//电流超限监测
FOR i:=1 TO g_maxCartJoint BY 1 DO
	m_checkDelay[i_armId].T_cartJntCurrentErr[i](IN:= ABS(i_cartJointData.m_curJntTrq[i])>g_cartMaxJntCurrent[i] AND m_checkPermit[i_ArmId].m_cartJntCurrentErr[i], PT:=m_checkDelayTime.Ti_CarJntCurrent , Q=> , ET=> );
	IF m_checkDelay[i_armId].T_cartJntCurrentErr[i].Q THEN
		errCodeAssign(i_armId, i_ArmId,  0, i, 16#2005 ,m_rcvLevel );
	END_IF
END_FOR


//Ethercat通讯检测
FOR i:=1 TO g_maxCartJoint BY 1 DO
	IF NOT i_safetyCheckVar.m_cartEtherCATState[i].EtherCATState THEN
		errCodeAssign(i_armId, i_ArmId,  0, i, 16#2006 ,m_rcvLevel );
	END_IF
END_FOR
END_METHOD

PROPERTY checkPermit : REFERENCE TO ARRAY[1..g_maxNum] OF  checkPermit
GET
checkPermit ref= m_checkPermit;
END_GET
SET
END_SET
END_PROPERTY

METHOD electriAngleDev : DINT
VAR_INPUT
	i_motorElectriAngleDev : DINT;
END_VAR

IF i_motorElectriAngleDev > 50000 THEN
	electriAngleDev := i_motorElectriAngleDev - 65535;
ELSIF i_motorElectriAngleDev < -50000 THEN
	electriAngleDev := i_motorElectriAngleDev + 65535;
ELSE
	electriAngleDev := i_motorElectriAngleDev;
END_IF
END_METHOD

METHOD errCodeAssign : BOOL
VAR_INPUT
	i_armId:UDINT;
	i_errLocation:UDINT;
	i_errCodeMode:UDINT;
	i_errJoint:UDINT;
	i_errID:UDINT;
	i_errFlagID :UINT;
END_VAR
IF m_jntErrFlag[i_armId,i_errJoint,i_errFlagID]=FALSE THEN
	m_jntErrFlag[i_armId,i_errJoint,i_errFlagID]:=TRUE;
	m_errCode:=SHL(i_errLocation,24)+SHL(i_errCodeMode,20)+SHL(i_errJoint,16)+i_errID;
	
	
	IF i_errID>=16#3000 THEN
		m_errNumType[m_unrcvLevel]:=LIMIT(0,m_errNumType[m_unrcvLevel]+1,100);
		m_arrayErrCodeType[m_unrcvLevel][m_errNumType[m_unrcvLevel]]:=m_errCode;
		g_arrayErrCodeArm[i_armId]:=arrayFILO(i_Array:= g_arrayErrCodeArm[i_ArmId], i_NewData:=m_errCode );
		m_armErrFlag[i_armId,m_unrcvLevel]:=TRUE;
		
	ELSIF i_errID>=16#2000 THEN
		m_errNumType[m_rcvLevel]:=LIMIT(0,m_errNumType[m_rcvLevel]+1,100);
		m_arrayErrCodeType[m_rcvLevel][m_errNumType[m_rcvLevel]]:=m_errCode;
		g_arrayErrCodeArm[i_armId]:=arrayFILO(i_Array:= g_arrayErrCodeArm[i_ArmId], i_NewData:=m_errCode );
		m_armErrFlag[i_armId,m_rcvLevel]:=TRUE;
		
	END_IF
END_IF
END_METHOD

METHOD errCodeUpdating :ARRAY [1..3] OF UDINT;
VAR_INPUT
END_VAR

m_errCodeUpdateTon[m_unrcvLevel](IN:= NOT m_errCodeUpdateFlag[3], PT:=m_codeUpdateDelay , Q=> m_errCodeUpdateFlag[3], ET=> );
IF m_errCodeUpdateFlag[m_unrcvLevel] THEN
	IF m_errNumType[m_unrcvLevel]>=1 THEN
		m_ArrayErrCodeType[m_unrcvLevel]:=ArrayDeleteFrist(i_Array:=m_ArrayErrCodeType[3]) ;
		o_ErrCode[m_unrcvLevel]:=m_ArrayErrCodeType[m_unrcvLevel][0] ;
		m_errNumType[m_unrcvLevel]:=m_errNumType[m_unrcvLevel]-1;
	END_IF
END_IF


m_errCodeUpdateTon[m_rcvLevel](IN:= NOT m_errCodeUpdateFlag[2], PT:=m_codeUpdateDelay , Q=> m_errCodeUpdateFlag[2], ET=> );
IF m_errCodeUpdateFlag[m_rcvLevel] THEN
	IF m_errNumType[m_rcvLevel]>=1 THEN
		m_ArrayErrCodeType[m_rcvLevel]:=ArrayDeleteFrist(i_Array:=m_ArrayErrCodeType[m_rcvLevel]) ;
		o_ErrCode[m_rcvLevel]:=m_ArrayErrCodeType[m_rcvLevel][0] ;
		m_errNumType[m_rcvLevel]:=m_errNumType[m_rcvLevel]-1;
	END_IF
END_IF
END_METHOD

METHOD errFlagReset : BOOL
VAR_INPUT
END_VAR

FOR i := 1 TO g_maxNum DO
	FOR j :=0 TO g_maxArmJoint DO
		m_jntErrFlag[i, j, 2]:=FALSE;
	END_FOR
	m_armErrFlag[i, 2]:=FALSE;
END_FOR

o_ErrCode[2]:=0;
END_METHOD

METHOD poseErrCheck : vec6d
VAR_INPUT
	i_cmdPose : ST_Frame;
	i_curPose :ST_Frame;
END_VAR

VAR
	posErr,oriErr:Vec3d;
	matT,rotErr:Mat3d;
	errAngle :LREAL;
	errAxis :Vec3d;
	i : INT;
END_VAR
vecSub(i_cmdPose.m_pos, i_curPose.m_pos,posErr);

matTranspose(i_cmdPose.m_rot, matT);
matMultiply(matT,i_curPose.m_rot, rotErr);
rot2AngAxis(rotErr, angle=>errAngle, axis=>errAxis);
vecMultiNum(errAxis, errAngle,oriErr);

FOR i := 1 TO 6 DO
	IF i <= 3 THEN
		poseErrCheck[i] := posErr[i];
	ELSE
		poseErrCheck[i] := oriErr[i];
	END_IF
END_FOR
END_METHOD

METHOD promptMassCode : BOOL
VAR_INPUT
	i_PromptStatus:BOOL;
	i_ArmId:UDINT;
	i_ErrID:UDINT;
	i_ErrLocation:UDINT;
END_VAR

m_PromptMassBusy:=TRUE;

//提示置位
IF i_PromptStatus=TRUE AND m_PromptFlag[i_ArmId,i_ErrID]=0 THEN
	m_PromptFlag[i_ArmId,i_ErrID]:=1;
END_IF

//输出提示故障码
IF m_PromptFlag[i_ArmId,i_ErrID]=1 THEN
	m_ErrCode:=SHL(i_ErrLocation,24)+i_ErrID+16#1010;
	m_ArrayErrCodeType[1]:=ArrayFIFO(i_Array:= m_ArrayErrCodeType[1], i_NewData:=m_ErrCode );//m_ErrCode;
	m_PromptFlag[i_ArmId,i_ErrID]:=2;
END_IF

//清除提示故障码
IF m_PromptFlag[i_ArmId,i_ErrID]=2 AND i_PromptStatus=FALSE THEN
	m_deleteCode:=SHL(i_ErrLocation,24)+i_ErrID+16#1010;
	ArrayDeleteInput(i_Array:= m_ArrayErrCodeType[1], i_DeleteCode:=m_deleteCode , o_Array=> m_ArrayErrCodeType[1]);
	m_PromptFlag[i_ArmId,i_ErrID]:=0;
END_IF
o_ErrCode[1]:=m_ArrayErrCodeType[1][0];
m_PromptMassBusy:=FALSE;
END_METHOD

METHOD systemSafetyCheck : BOOL
VAR_INPUT
	i_armId:UDINT;
	i_safetyCheckVar :ARRAY[1..g_maxNum] OF checkInputVariable;
	i_masterStatus :ST_MasterStatus;
	i_cartJointData : ST_CartJointData;
	i_masterJointData : ST_MasterJointData;
END_VAR

VAR
	k:INT;
END_VAR
IF i_armId =g_cartNum THEN 
	//cart safrty check
	cartSafetyCheck(i_armId,i_safetyCheckVar[i_armId],i_cartJointData);
ELSE
	//master arms safety check
	armSafetyCheck(i_armId,i_safetyCheckVar,i_masterStatus,i_masterJointData);
END_IF

//StopButton
IF  i_safetyCheckVar[i_ArmId].PCStopButton=0 OR NOT i_safetyCheckVar[i_ArmId].MasterStopButton OR i_safetyCheckVar[i_ArmId].SlaveStopButton THEN
	errCodeAssign(i_ArmId, 16#0B, 0, 0, 16#2001, m_rcvLevel );
END_IF

//prompt message
FOR i:=1 TO 10 DO
	PromptMassCode( i_safetyCheckVar[i_ArmId].m_promptStatus[i], i_ArmId,  i,  i_safetyCheckVar[i_ArmId].m_promptLocation[i]);
END_FOR
END_METHOD

END_FUNCTION_BLOCK

// ---- SafetyCheck/Fb_dataRecord.TcPOU
FUNCTION_BLOCK Fb_dataRecord 
VAR_INPUT
	
END_VAR
VAR_OUTPUT
END_VAR
VAR
	i,j,k,z,c:UDINT;
	Index:ARRAY[1..g_maxNum] OF INT:=[3(2)];
	m_Index:ARRAY[1..g_maxNum] OF UDINT;
	Err,Arm,Joint,ErrID:UDINT;
	ErrWritingFalg:ARRAY [1..g_maxNum] OF BOOL:=[3(FALSE)];
	ArrayErrCodeTypeLast:ARRAY [1..g_maxNum] OF UDINT;
	sPath: STRING(255);
	mErr:ARRAY [0..MAX_CSV_COLUMNS] OF STRING(255);
	StartRecord:ARRAY[1..g_maxNum] OF R_TRIG;
	RecordCompletion:ARRAY[1..g_maxNum] OF F_TRIG;
	errFlagDelay1s : ARRAY [1..3] OF TON;
	errWritingAllowed : ARRAY [1..3] OF BOOL:=[3(FALSE)];
	
	fbSysTime	: 	GETSYSTEMTIME;
	tFileTime	:	T_FILETIME;  
	
	_tNow,	_tNowBoLin	:	TIMESTRUCT; 
	fbFormat 	: 	FB_FormatString;
	_sPathFormat	: T_MaxString := '%s%d-%d-%d-%d-%d-%d-%s-%s-%s.csv'; 
	
	_iBuffer: UDINT := 1;
		
	StartTime:LREAL;
	
	iZeroRowsData:ARRAY[0..MAX_CSV_ROWS] OF  ARRAY [0..MAX_CSV_COLUMNS] OF STRING(MAX_CSV_FIELD_LENGTH);
	iZeroErrCode:ARRAY [1..g_maxNum] OF ARRAY[0..100] OF UDINT;
	gCSV_Buffer: ARRAY[1..MAX_CSV_RING_BUFFER] OF ST_Buffer;
	mErrNameLocation: ARRAY [1..MAX_CSV_RING_BUFFER,0..MAX_CSV_COLUMNS] OF STRING(MAX_CSV_FIELD_LENGTH);
END_VAR

METHOD armDataCast : BOOL
VAR_IN_OUT CONSTANT
	i_safetyCheckVar :ARRAY[1..g_maxNum] OF checkInputVariable;
	i_masterStatus : ST_masterStatus;
	i_masterJointData : ST_MasterJointData;
END_VAR

FOR i:= 1 TO 2 BY 1 DO
	IF ErrWritingFalg[i] = FALSE THEN
	j:=1;
	//状态机
	gCSV_Buffer[i].aBuffer[Index[i]][j:=j+1]:=LREAL_TO_FMTSTR(i_masterStatus.m_armState[i],0, TRUE);  gCSV_Buffer[i].aBuffer[1][j]:='armMachine';
	
	//link pos
	gCSV_Buffer[i].aBuffer[Index[i]][j:=j+1]:=LREAL_TO_STRING(i_masterJointData.m_curLinkPos[i][1]);   gCSV_Buffer[i].aBuffer[1][j]:='curLinkPosJ1';
	gCSV_Buffer[i].aBuffer[Index[i]][j:=j+1]:=LREAL_TO_STRING(i_masterJointData.m_curLinkPos[i][2]);   gCSV_Buffer[i].aBuffer[1][j]:='curLinkPosJ2';
	gCSV_Buffer[i].aBuffer[Index[i]][j:=j+1]:=LREAL_TO_STRING(i_masterJointData.m_curLinkPos[i][3]);   gCSV_Buffer[i].aBuffer[1][j]:='curLinkPosJ3';
	gCSV_Buffer[i].aBuffer[Index[i]][j:=j+1]:=LREAL_TO_STRING(i_masterJointData.m_curLinkPos[i][4]);   gCSV_Buffer[i].aBuffer[1][j]:='curLinkPosJ4';
	gCSV_Buffer[i].aBuffer[Index[i]][j:=j+1]:=LREAL_TO_STRING(i_masterJointData.m_curLinkPos[i][5]);   gCSV_Buffer[i].aBuffer[1][j]:='curLinkPosJ5';
	gCSV_Buffer[i].aBuffer[Index[i]][j:=j+1]:=LREAL_TO_STRING(i_masterJointData.m_curLinkPos[i][6]);   gCSV_Buffer[i].aBuffer[1][j]:='curLinkPosJ6';
	gCSV_Buffer[i].aBuffer[Index[i]][j:=j+1]:=LREAL_TO_STRING(i_masterJointData.m_curLinkPos[i][7]);   gCSV_Buffer[i].aBuffer[1][j]:='curLinkPosJ7';
	
	//motor pos / curJntPos
	gCSV_Buffer[i].aBuffer[Index[i]][j:=j+1]:=LREAL_TO_STRING(i_masterJointData.m_curJntPos[i][1]);  gCSV_Buffer[i].aBuffer[1][j]:='curJntPosJ1';
	gCSV_Buffer[i].aBuffer[Index[i]][j:=j+1]:=LREAL_TO_STRING(i_masterJointData.m_curJntPos[i][2]);  gCSV_Buffer[i].aBuffer[1][j]:='curJntPosJ2';
	gCSV_Buffer[i].aBuffer[Index[i]][j:=j+1]:=LREAL_TO_STRING(i_masterJointData.m_curJntPos[i][3]);  gCSV_Buffer[i].aBuffer[1][j]:='curJntPosJ3';
	gCSV_Buffer[i].aBuffer[Index[i]][j:=j+1]:=LREAL_TO_STRING(i_masterJointData.m_curJntPos[i][4]);  gCSV_Buffer[i].aBuffer[1][j]:='curJntPosJ4';
	gCSV_Buffer[i].aBuffer[Index[i]][j:=j+1]:=LREAL_TO_STRING(i_masterJointData.m_curJntPos[i][5]); 	gCSV_Buffer[i].aBuffer[1][j]:='curJntPosJ5';
	gCSV_Buffer[i].aBuffer[Index[i]][j:=j+1]:=LREAL_TO_STRING(i_masterJointData.m_curJntPos[i][6]); 	gCSV_Buffer[i].aBuffer[1][j]:='curJntPosJ6';
	gCSV_Buffer[i].aBuffer[Index[i]][j:=j+1]:=LREAL_TO_STRING(i_masterJointData.m_curJntPos[i][7]); 	gCSV_Buffer[i].aBuffer[1][j]:='curJntPosJ7';
	
	
	//target joint position 
	gCSV_Buffer[i].aBuffer[Index[i]][j:=j+1]:=LREAL_TO_STRING(i_masterJointData.m_cmdJntPos[i][1]);  gCSV_Buffer[i].aBuffer[1][j]:='cmdJntPosJ1';
	gCSV_Buffer[i].aBuffer[Index[i]][j:=j+1]:=LREAL_TO_STRING(i_masterJointData.m_cmdJntPos[i][2]);  gCSV_Buffer[i].aBuffer[1][j]:='cmdJntPosJ2';
	gCSV_Buffer[i].aBuffer[Index[i]][j:=j+1]:=LREAL_TO_STRING(i_masterJointData.m_cmdJntPos[i][3]);  gCSV_Buffer[i].aBuffer[1][j]:='cmdJntPosJ3';
	gCSV_Buffer[i].aBuffer[Index[i]][j:=j+1]:=LREAL_TO_STRING(i_masterJointData.m_cmdJntPos[i][4]);  gCSV_Buffer[i].aBuffer[1][j]:='cmdJntPosJ4';
	gCSV_Buffer[i].aBuffer[Index[i]][j:=j+1]:=LREAL_TO_STRING(i_masterJointData.m_cmdJntPos[i][5]);  gCSV_Buffer[i].aBuffer[1][j]:='cmdJntPosJ5';
	gCSV_Buffer[i].aBuffer[Index[i]][j:=j+1]:=LREAL_TO_STRING(i_masterJointData.m_cmdJntPos[i][6]);  gCSV_Buffer[i].aBuffer[1][j]:='cmdJntPosJ6';
	gCSV_Buffer[i].aBuffer[Index[i]][j:=j+1]:=LREAL_TO_STRING(i_masterJointData.m_cmdJntPos[i][7]);  gCSV_Buffer[i].aBuffer[1][j]:='cmdJntPosJ7';
	
	
	//current joint velocity
	gCSV_Buffer[i].aBuffer[Index[i]][j:=j+1]:=LREAL_TO_STRING(i_masterJointData.m_curJntVel[i][1]);  gCSV_Buffer[i].aBuffer[1][j]:='curJntVelJ1';
	gCSV_Buffer[i].aBuffer[Index[i]][j:=j+1]:=LREAL_TO_STRING(i_masterJointData.m_curJntVel[i][2]);  gCSV_Buffer[i].aBuffer[1][j]:='curJntVelJ2';
	gCSV_Buffer[i].aBuffer[Index[i]][j:=j+1]:=LREAL_TO_STRING(i_masterJointData.m_curJntVel[i][3]);  gCSV_Buffer[i].aBuffer[1][j]:='curJntVelJ3';
	gCSV_Buffer[i].aBuffer[Index[i]][j:=j+1]:=LREAL_TO_STRING(i_masterJointData.m_curJntVel[i][4]);  gCSV_Buffer[i].aBuffer[1][j]:='curJntVelJ4';
	gCSV_Buffer[i].aBuffer[Index[i]][j:=j+1]:=LREAL_TO_STRING(i_masterJointData.m_curJntVel[i][5]);  gCSV_Buffer[i].aBuffer[1][j]:='curJntVelJ5';
	gCSV_Buffer[i].aBuffer[Index[i]][j:=j+1]:=LREAL_TO_STRING(i_masterJointData.m_curJntVel[i][6]);  gCSV_Buffer[i].aBuffer[1][j]:='curJntVelJ6';
	gCSV_Buffer[i].aBuffer[Index[i]][j:=j+1]:=LREAL_TO_STRING(i_masterJointData.m_curJntVel[i][7]);  gCSV_Buffer[i].aBuffer[1][j]:='curJntVelJ7';
	
	//command arm pose
	gCSV_Buffer[i].aBuffer[Index[i]][j:=j+1]:=LREAL_TO_STRING(i_masterStatus.m_cmdArmPose[i].m_pos[1]);  gCSV_Buffer[i].aBuffer[1][j]:='cmdArmPose1';
	gCSV_Buffer[i].aBuffer[Index[i]][j:=j+1]:=LREAL_TO_STRING(i_masterStatus.m_cmdArmPose[i].m_pos[2]);  gCSV_Buffer[i].aBuffer[1][j]:='cmdArmPose2';
	gCSV_Buffer[i].aBuffer[Index[i]][j:=j+1]:=LREAL_TO_STRING(i_masterStatus.m_cmdArmPose[i].m_pos[3]);  gCSV_Buffer[i].aBuffer[1][j]:='cmdArmPose3';
	//gCSV_Buffer[i].aBuffer[Index[i]][j:=j+1]:=LREAL_TO_STRING(i_masterStatus.m_cmdArmPose[i].m_rot[1]);   gCSV_Buffer[i].aBuffer[1][j]:='cmdArmPose4';
	//gCSV_Buffer[i].aBuffer[Index[i]][j:=j+1]:=LREAL_TO_STRING(i_masterStatus.m_cmdArmPose[i].m_rot[2]);   gCSV_Buffer[i].aBuffer[1][j]:='cmdArmPose5';
	//gCSV_Buffer[i].aBuffer[Index[i]][j:=j+1]:=LREAL_TO_STRING(i_masterStatus.m_cmdArmPose[i].m_rot[3]);   gCSV_Buffer[i].aBuffer[1][j]:='cmdArmPose6';

	//current arm pose
	gCSV_Buffer[i].aBuffer[Index[i]][j:=j+1]:=LREAL_TO_STRING(i_masterStatus.m_curArmPose[i].m_pos[1]);  gCSV_Buffer[i].aBuffer[1][j]:='curArmPose1';
	gCSV_Buffer[i].aBuffer[Index[i]][j:=j+1]:=LREAL_TO_STRING(i_masterStatus.m_curArmPose[i].m_pos[2]);  gCSV_Buffer[i].aBuffer[1][j]:='curArmPose2';
	gCSV_Buffer[i].aBuffer[Index[i]][j:=j+1]:=LREAL_TO_STRING(i_masterStatus.m_curArmPose[i].m_pos[3]);  gCSV_Buffer[i].aBuffer[1][j]:='curArmPose3';
	//gCSV_Buffer[i].aBuffer[Index[i]][j:=j+1]:=LREAL_TO_STRING(i_masterStatus.m_curArmPose[i].m_rot[1]);   gCSV_Buffer[i].aBuffer[1][j]:='curArmPose4';
	//gCSV_Buffer[i].aBuffer[Index[i]][j:=j+1]:=LREAL_TO_STRING(i_masterStatus.m_curArmPose[i].m_rot[2]);   gCSV_Buffer[i].aBuffer[1][j]:='curArmPose5';
	//gCSV_Buffer[i].aBuffer[Index[i]][j:=j+1]:=LREAL_TO_STRING(i_masterStatus.m_curArmPose[i].m_rot[3]);   gCSV_Buffer[i].aBuffer[1][j]:='curArmPose6';
	
	//drive error word
	gCSV_Buffer[i].aBuffer[Index[i]][j:=j+1]:=UDINT_TO_STRING(i_safetyCheckVar[i].m_masterDriverInput[1].m_driverError);  gCSV_Buffer[i].aBuffer[1][j]:='driverErrorIOJ1'; 
	gCSV_Buffer[i].aBuffer[Index[i]][j:=j+1]:=UDINT_TO_STRING(i_safetyCheckVar[i].m_masterDriverInput[2].m_driverError);  gCSV_Buffer[i].aBuffer[1][j]:='driverErrorIOJ2'; 
	gCSV_Buffer[i].aBuffer[Index[i]][j:=j+1]:=UDINT_TO_STRING(i_safetyCheckVar[i].m_masterDriverInput[3].m_driverError);  gCSV_Buffer[i].aBuffer[1][j]:='driverErrorIOJ3'; 
	gCSV_Buffer[i].aBuffer[Index[i]][j:=j+1]:=UDINT_TO_STRING(i_safetyCheckVar[i].m_masterDriverInput[4].m_driverError);  gCSV_Buffer[i].aBuffer[1][j]:='driverErrorIOJ4'; 
	gCSV_Buffer[i].aBuffer[Index[i]][j:=j+1]:=UDINT_TO_STRING(i_safetyCheckVar[i].m_masterDriverInput[5].m_driverError); gCSV_Buffer[i].aBuffer[1][j]:='driverErrorIOJ5'; 
	gCSV_Buffer[i].aBuffer[Index[i]][j:=j+1]:=UDINT_TO_STRING(i_safetyCheckVar[i].m_masterDriverInput[6].m_driverError); gCSV_Buffer[i].aBuffer[1][j]:='driverErrorIOJ6'; 
	gCSV_Buffer[i].aBuffer[Index[i]][j:=j+1]:=UDINT_TO_STRING(i_safetyCheckVar[i].m_masterDriverInput[7].m_driverError); gCSV_Buffer[i].aBuffer[1][j]:='driverErrorIOJ7'; 
   
	
	//link encoder IO
	gCSV_Buffer[i].aBuffer[Index[i]][j:=j+1]:=DINT_TO_STRING(i_safetyCheckVar[i].m_masterDriverInput[1].m_linkEncoder);  gCSV_Buffer[i].aBuffer[1][j]:='curLinkIOJ1';
	gCSV_Buffer[i].aBuffer[Index[i]][j:=j+1]:=DINT_TO_STRING(i_safetyCheckVar[i].m_masterDriverInput[2].m_linkEncoder);  gCSV_Buffer[i].aBuffer[1][j]:='curLinkIOJ2';
	gCSV_Buffer[i].aBuffer[Index[i]][j:=j+1]:=DINT_TO_STRING(i_safetyCheckVar[i].m_masterDriverInput[3].m_linkEncoder);  gCSV_Buffer[i].aBuffer[1][j]:='curLinkIOJ3';
	gCSV_Buffer[i].aBuffer[Index[i]][j:=j+1]:=DINT_TO_STRING(i_safetyCheckVar[i].m_masterDriverInput[4].m_linkEncoder);  gCSV_Buffer[i].aBuffer[1][j]:='curLinkIOJ4';
	gCSV_Buffer[i].aBuffer[Index[i]][j:=j+1]:=DINT_TO_STRING(i_safetyCheckVar[i].m_masterDriverInput[5].m_linkEncoder);  gCSV_Buffer[i].aBuffer[1][j]:='curLinkIOJ5';
	gCSV_Buffer[i].aBuffer[Index[i]][j:=j+1]:=DINT_TO_STRING(i_safetyCheckVar[i].m_masterDriverInput[6].m_linkEncoder);  gCSV_Buffer[i].aBuffer[1][j]:='curLinkIOJ6';
	gCSV_Buffer[i].aBuffer[Index[i]][j:=j+1]:=DINT_TO_STRING(i_safetyCheckVar[i].m_masterDriverInput[7].m_linkEncoder);  gCSV_Buffer[i].aBuffer[1][j]:='curLinkIOJ7';
	
	//motor encoder  IO
	gCSV_Buffer[i].aBuffer[Index[i]][j:=j+1]:=DINT_TO_STRING(i_safetyCheckVar[i].m_masterDriverInput[1].m_motorEncoder);  gCSV_Buffer[i].aBuffer[1][j]:='curMotorEncIOJ1';
	gCSV_Buffer[i].aBuffer[Index[i]][j:=j+1]:=DINT_TO_STRING(i_safetyCheckVar[i].m_masterDriverInput[2].m_motorEncoder);  gCSV_Buffer[i].aBuffer[1][j]:='curMotorEncIOJ2';
	gCSV_Buffer[i].aBuffer[Index[i]][j:=j+1]:=DINT_TO_STRING(i_safetyCheckVar[i].m_masterDriverInput[3].m_motorEncoder);  gCSV_Buffer[i].aBuffer[1][j]:='curMotorEncIOJ3';
	gCSV_Buffer[i].aBuffer[Index[i]][j:=j+1]:=DINT_TO_STRING(i_safetyCheckVar[i].m_masterDriverInput[4].m_motorEncoder);  gCSV_Buffer[i].aBuffer[1][j]:='curMotorEncIOJ4';
	gCSV_Buffer[i].aBuffer[Index[i]][j:=j+1]:=DINT_TO_STRING(i_safetyCheckVar[i].m_masterDriverInput[5].m_motorEncoder);  gCSV_Buffer[i].aBuffer[1][j]:='curMotorEncIOJ5';
	gCSV_Buffer[i].aBuffer[Index[i]][j:=j+1]:=DINT_TO_STRING(i_safetyCheckVar[i].m_masterDriverInput[6].m_motorEncoder);  gCSV_Buffer[i].aBuffer[1][j]:='curMotorEncIOJ6';
	gCSV_Buffer[i].aBuffer[Index[i]][j:=j+1]:=DINT_TO_STRING(i_safetyCheckVar[i].m_masterDriverInput[7].m_motorEncoder);  gCSV_Buffer[i].aBuffer[1][j]:='curMotorEncIOJ7';
	
	//status word IO
	gCSV_Buffer[i].aBuffer[Index[i]][j:=j+1]:=UINT_TO_STRING(i_safetyCheckVar[i].m_masterDriverInput[1].m_statusWord);	gCSV_Buffer[i].aBuffer[1][j]:='statusWordIOJ1';
	gCSV_Buffer[i].aBuffer[Index[i]][j:=j+1]:=UINT_TO_STRING(i_safetyCheckVar[i].m_masterDriverInput[2].m_statusWord);	gCSV_Buffer[i].aBuffer[1][j]:='statusWordIOJ2';
	gCSV_Buffer[i].aBuffer[Index[i]][j:=j+1]:=UINT_TO_STRING(i_safetyCheckVar[i].m_masterDriverInput[3].m_statusWord);	gCSV_Buffer[i].aBuffer[1][j]:='statusWordIOJ3';
	gCSV_Buffer[i].aBuffer[Index[i]][j:=j+1]:=UINT_TO_STRING(i_safetyCheckVar[i].m_masterDriverInput[4].m_statusWord);	gCSV_Buffer[i].aBuffer[1][j]:='statusWordIOJ4';
	gCSV_Buffer[i].aBuffer[Index[i]][j:=j+1]:=UINT_TO_STRING(i_safetyCheckVar[i].m_masterDriverInput[5].m_statusWord);	gCSV_Buffer[i].aBuffer[1][j]:='statusWordIOJ5';
	gCSV_Buffer[i].aBuffer[Index[i]][j:=j+1]:=UINT_TO_STRING(i_safetyCheckVar[i].m_masterDriverInput[6].m_statusWord);	gCSV_Buffer[i].aBuffer[1][j]:='statusWordIOJ6';
	gCSV_Buffer[i].aBuffer[Index[i]][j:=j+1]:=UINT_TO_STRING(i_safetyCheckVar[i].m_masterDriverInput[7].m_statusWord);	gCSV_Buffer[i].aBuffer[1][j]:='statusWordIOJ7';

	//current torque IO
	gCSV_Buffer[i].aBuffer[Index[i]][j:=j+1]:=DINT_TO_STRING(i_safetyCheckVar[i].m_masterDriverInput[1].m_current);  gCSV_Buffer[i].aBuffer[1][j]:='curTorqueIOJ1';
	gCSV_Buffer[i].aBuffer[Index[i]][j:=j+1]:=DINT_TO_STRING(i_safetyCheckVar[i].m_masterDriverInput[2].m_current);  gCSV_Buffer[i].aBuffer[1][j]:='curTorqueIOJ2';
	gCSV_Buffer[i].aBuffer[Index[i]][j:=j+1]:=DINT_TO_STRING(i_safetyCheckVar[i].m_masterDriverInput[3].m_current);  gCSV_Buffer[i].aBuffer[1][j]:='curTorqueIOJ3';
	gCSV_Buffer[i].aBuffer[Index[i]][j:=j+1]:=DINT_TO_STRING(i_safetyCheckVar[i].m_masterDriverInput[4].m_current);  gCSV_Buffer[i].aBuffer[1][j]:='curTorqueIOJ4';
	gCSV_Buffer[i].aBuffer[Index[i]][j:=j+1]:=DINT_TO_STRING(i_safetyCheckVar[i].m_masterDriverInput[5].m_current);  gCSV_Buffer[i].aBuffer[1][j]:='curTorqueIOJ5';
	gCSV_Buffer[i].aBuffer[Index[i]][j:=j+1]:=DINT_TO_STRING(i_safetyCheckVar[i].m_masterDriverInput[6].m_current);  gCSV_Buffer[i].aBuffer[1][j]:='curTorqueIOJ6';
	gCSV_Buffer[i].aBuffer[Index[i]][j:=j+1]:=DINT_TO_STRING(i_safetyCheckVar[i].m_masterDriverInput[7].m_current);  gCSV_Buffer[i].aBuffer[1][j]:='curTorqueIOJ7';
	
	//target torque IO
	gCSV_Buffer[i].aBuffer[Index[i]][j:=j+1]:=DINT_TO_STRING(i_safetyCheckVar[i].m_masterDriverOutput[1].m_cmdCurrent);  gCSV_Buffer[i].aBuffer[1][j]:='cmdTorqueIOJ1';
	gCSV_Buffer[i].aBuffer[Index[i]][j:=j+1]:=DINT_TO_STRING(i_safetyCheckVar[i].m_masterDriverOutput[2].m_cmdCurrent);  gCSV_Buffer[i].aBuffer[1][j]:='cmdTorqueIOJ2';
	gCSV_Buffer[i].aBuffer[Index[i]][j:=j+1]:=DINT_TO_STRING(i_safetyCheckVar[i].m_masterDriverOutput[3].m_cmdCurrent);  gCSV_Buffer[i].aBuffer[1][j]:='cmdTorqueIOJ3';
	gCSV_Buffer[i].aBuffer[Index[i]][j:=j+1]:=DINT_TO_STRING(i_safetyCheckVar[i].m_masterDriverOutput[4].m_cmdCurrent);  gCSV_Buffer[i].aBuffer[1][j]:='cmdTorqueIOJ4';
	gCSV_Buffer[i].aBuffer[Index[i]][j:=j+1]:=DINT_TO_STRING(i_safetyCheckVar[i].m_masterDriverOutput[5].m_cmdCurrent);  gCSV_Buffer[i].aBuffer[1][j]:='cmdTorqueIOJ5';
	gCSV_Buffer[i].aBuffer[Index[i]][j:=j+1]:=DINT_TO_STRING(i_safetyCheckVar[i].m_masterDriverOutput[6].m_cmdCurrent);  gCSV_Buffer[i].aBuffer[1][j]:='cmdTorqueIOJ6';
	gCSV_Buffer[i].aBuffer[Index[i]][j:=j+1]:=DINT_TO_STRING(i_safetyCheckVar[i].m_masterDriverOutput[7].m_cmdCurrent);  gCSV_Buffer[i].aBuffer[1][j]:='cmdTorqueIOJ7';
	
	//target motor encoder IO
	gCSV_Buffer[i].aBuffer[Index[i]][j:=j+1]:=DINT_TO_STRING(i_safetyCheckVar[i].m_masterDriverOutput[1].m_cmdMotorEncoder);  gCSV_Buffer[i].aBuffer[1][j]:='cmdMotorEncIOJ1';
	gCSV_Buffer[i].aBuffer[Index[i]][j:=j+1]:=DINT_TO_STRING(i_safetyCheckVar[i].m_masterDriverOutput[2].m_cmdMotorEncoder);  gCSV_Buffer[i].aBuffer[1][j]:='cmdMotorEncIOJ2';
	gCSV_Buffer[i].aBuffer[Index[i]][j:=j+1]:=DINT_TO_STRING(i_safetyCheckVar[i].m_masterDriverOutput[3].m_cmdMotorEncoder);  gCSV_Buffer[i].aBuffer[1][j]:='cmdMotorEncIOJ3';
	gCSV_Buffer[i].aBuffer[Index[i]][j:=j+1]:=DINT_TO_STRING(i_safetyCheckVar[i].m_masterDriverOutput[4].m_cmdMotorEncoder);  gCSV_Buffer[i].aBuffer[1][j]:='cmdMotorEncIOJ4';
	gCSV_Buffer[i].aBuffer[Index[i]][j:=j+1]:=DINT_TO_STRING(i_safetyCheckVar[i].m_masterDriverOutput[5].m_cmdMotorEncoder);  gCSV_Buffer[i].aBuffer[1][j]:='cmdMotorEncIOJ5';
	gCSV_Buffer[i].aBuffer[Index[i]][j:=j+1]:=DINT_TO_STRING(i_safetyCheckVar[i].m_masterDriverOutput[6].m_cmdMotorEncoder);  gCSV_Buffer[i].aBuffer[1][j]:='cmdMotorEncIOJ6';
	gCSV_Buffer[i].aBuffer[Index[i]][j:=j+1]:=DINT_TO_STRING(i_safetyCheckVar[i].m_masterDriverOutput[7].m_cmdMotorEncoder);  gCSV_Buffer[i].aBuffer[1][j]:='cmdMotorEncIOJ7';


	//output motor opMode IO
	gCSV_Buffer[i].aBuffer[Index[i]][j:=j+1]:=DINT_TO_STRING(i_safetyCheckVar[i].m_masterDriverOutput[1].m_opMode);  gCSV_Buffer[i].aBuffer[1][j]:='opModeIOJ1';
	gCSV_Buffer[i].aBuffer[Index[i]][j:=j+1]:=DINT_TO_STRING(i_safetyCheckVar[i].m_masterDriverOutput[2].m_opMode);  gCSV_Buffer[i].aBuffer[1][j]:='opModeIOJ2';
	gCSV_Buffer[i].aBuffer[Index[i]][j:=j+1]:=DINT_TO_STRING(i_safetyCheckVar[i].m_masterDriverOutput[3].m_opMode);  gCSV_Buffer[i].aBuffer[1][j]:='opModeIOJ3';
	gCSV_Buffer[i].aBuffer[Index[i]][j:=j+1]:=DINT_TO_STRING(i_safetyCheckVar[i].m_masterDriverOutput[4].m_opMode);  gCSV_Buffer[i].aBuffer[1][j]:='opModeIOJ4';
	gCSV_Buffer[i].aBuffer[Index[i]][j:=j+1]:=DINT_TO_STRING(i_safetyCheckVar[i].m_masterDriverOutput[5].m_opMode);  gCSV_Buffer[i].aBuffer[1][j]:='opModeIOJ5';
	gCSV_Buffer[i].aBuffer[Index[i]][j:=j+1]:=DINT_TO_STRING(i_safetyCheckVar[i].m_masterDriverOutput[6].m_opMode);  gCSV_Buffer[i].aBuffer[1][j]:='opModeIOJ6';
	gCSV_Buffer[i].aBuffer[Index[i]][j:=j+1]:=DINT_TO_STRING(i_safetyCheckVar[i].m_masterDriverOutput[7].m_opMode);  gCSV_Buffer[i].aBuffer[1][j]:='opModeIOJ7';

	END_IF
END_FOR
END_METHOD

METHOD cartDataCast : BOOL
VAR_IN_OUT CONSTANT
	i_safetyCheckVar : checkInputVariable;
	i_cartStatus : ST_CartStatus;
	i_cartJointData : ST_CartJointData;
END_VAR


IF ErrWritingFalg[3] = FALSE THEN
	c:=1;
	//cart Joint link position
	gCSV_Buffer[3].aBuffer[Index[3]][c:=c+1]:=LREAL_TO_STRING(i_cartJointData.m_curLinkPos[1]);  gCSV_Buffer[3].aBuffer[1][c]:='cartCurLinkPosJ1';
	gCSV_Buffer[3].aBuffer[Index[3]][c:=c+1]:=LREAL_TO_STRING(i_cartJointData.m_curLinkPos[2]);  gCSV_Buffer[3].aBuffer[1][c]:='cartCurLinkPosJ2';
	gCSV_Buffer[3].aBuffer[Index[3]][c:=c+1]:=LREAL_TO_STRING(i_cartJointData.m_curLinkPos[3]);  gCSV_Buffer[3].aBuffer[1][c]:='cartCurLinkPosJ3';
	gCSV_Buffer[3].aBuffer[Index[3]][c:=c+1]:=LREAL_TO_STRING(i_cartJointData.m_curLinkPos[4]);  gCSV_Buffer[3].aBuffer[1][c]:='cartCurLinkPosJ4';

	//cart current joint postion
	gCSV_Buffer[3].aBuffer[Index[3]][c:=c+1]:=LREAL_TO_STRING(i_cartJointData.m_curJntPos[1]);  gCSV_Buffer[3].aBuffer[1][c]:='curJntPosJ1';
	gCSV_Buffer[3].aBuffer[Index[3]][c:=c+1]:=LREAL_TO_STRING(i_cartJointData.m_curJntPos[2]);  gCSV_Buffer[3].aBuffer[1][c]:='curJntPosJ2';
	gCSV_Buffer[3].aBuffer[Index[3]][c:=c+1]:=LREAL_TO_STRING(i_cartJointData.m_curJntPos[3]);  gCSV_Buffer[3].aBuffer[1][c]:='curJntPosJ3';
	gCSV_Buffer[3].aBuffer[Index[3]][c:=c+1]:=LREAL_TO_STRING(i_cartJointData.m_curJntPos[4]);  gCSV_Buffer[3].aBuffer[1][c]:='curJntPosJ4';
	
	//cart target joint postion
	gCSV_Buffer[3].aBuffer[Index[3]][c:=c+1]:=LREAL_TO_STRING(i_cartJointData.m_cmdJntPos[1]);  gCSV_Buffer[3].aBuffer[1][c]:='cmdJntPosJ1';
	gCSV_Buffer[3].aBuffer[Index[3]][c:=c+1]:=LREAL_TO_STRING(i_cartJointData.m_cmdJntPos[2]);  gCSV_Buffer[3].aBuffer[1][c]:='cmdJntPosJ2';
	gCSV_Buffer[3].aBuffer[Index[3]][c:=c+1]:=LREAL_TO_STRING(i_cartJointData.m_cmdJntPos[3]);  gCSV_Buffer[3].aBuffer[1][c]:='cmdJntPosJ3';
	gCSV_Buffer[3].aBuffer[Index[3]][c:=c+1]:=LREAL_TO_STRING(i_cartJointData.m_cmdJntPos[4]);  gCSV_Buffer[3].aBuffer[1][c]:='cmdJntPosJ4';
	
	//drive error word
	gCSV_Buffer[3].aBuffer[Index[3]][c:=c+1]:=LREAL_TO_STRING(i_safetyCheckVar.m_cartDriverInput[1].m_driverError);  gCSV_Buffer[3].aBuffer[1][c]:='driverErrorJ1';
	gCSV_Buffer[3].aBuffer[Index[3]][c:=c+1]:=LREAL_TO_STRING(i_safetyCheckVar.m_cartDriverInput[2].m_driverError);  gCSV_Buffer[3].aBuffer[1][c]:='driverErrorJ2';
	gCSV_Buffer[3].aBuffer[Index[3]][c:=c+1]:=LREAL_TO_STRING(i_safetyCheckVar.m_cartDriverInput[3].m_driverError);  gCSV_Buffer[3].aBuffer[1][c]:='driverErrorJ3';
	gCSV_Buffer[3].aBuffer[Index[3]][c:=c+1]:=LREAL_TO_STRING(i_safetyCheckVar.m_cartDriverInput[4].m_driverError);  gCSV_Buffer[3].aBuffer[1][c]:='driverErrorJ4';
	
	//cart link encoder
	gCSV_Buffer[3].aBuffer[Index[3]][c:=c+1]:=LREAL_TO_STRING(i_safetyCheckVar.m_cartDriverInput[1].m_linkEncoder);  gCSV_Buffer[3].aBuffer[1][c]:='cartLinkIOJ1';
	gCSV_Buffer[3].aBuffer[Index[3]][c:=c+1]:=LREAL_TO_STRING(i_safetyCheckVar.m_cartDriverInput[2].m_linkEncoder);  gCSV_Buffer[3].aBuffer[1][c]:='cartLinkIOJ2';
	gCSV_Buffer[3].aBuffer[Index[3]][c:=c+1]:=LREAL_TO_STRING(i_safetyCheckVar.m_cartDriverInput[3].m_linkEncoder);  gCSV_Buffer[3].aBuffer[1][c]:='cartLinkIOJ3';
	gCSV_Buffer[3].aBuffer[Index[3]][c:=c+1]:=LREAL_TO_STRING(i_safetyCheckVar.m_cartDriverInput[4].m_linkEncoder);  gCSV_Buffer[3].aBuffer[1][c]:='cartLinkIOJ4';
	
	//cart actual torque 
	gCSV_Buffer[3].aBuffer[Index[3]][c:=c+1]:=DINT_TO_STRING(i_safetyCheckVar.m_cartDriverInput[1].m_current);  gCSV_Buffer[3].aBuffer[1][c]:='cartCurrentIOJ1';
	gCSV_Buffer[3].aBuffer[Index[3]][c:=c+1]:=DINT_TO_STRING(i_safetyCheckVar.m_cartDriverInput[2].m_current);  gCSV_Buffer[3].aBuffer[1][c]:='cartCurrentIOJ2';
	gCSV_Buffer[3].aBuffer[Index[3]][c:=c+1]:=DINT_TO_STRING(i_safetyCheckVar.m_cartDriverInput[3].m_current);  gCSV_Buffer[3].aBuffer[1][c]:='cartCurrentIOJ3';
	gCSV_Buffer[3].aBuffer[Index[3]][c:=c+1]:=DINT_TO_STRING(i_safetyCheckVar.m_cartDriverInput[4].m_current);  gCSV_Buffer[3].aBuffer[1][c]:='cartCurrentIOJ4';
		
	//cart joint status word
	gCSV_Buffer[3].aBuffer[Index[3]][c:=c+1]:=DINT_TO_STRING(i_safetyCheckVar.m_cartDriverInput[1].m_statusWord);  gCSV_Buffer[3].aBuffer[1][c]:='cartStatusWordIOJ1';
	gCSV_Buffer[3].aBuffer[Index[3]][c:=c+1]:=DINT_TO_STRING(i_safetyCheckVar.m_cartDriverInput[2].m_statusWord);  gCSV_Buffer[3].aBuffer[1][c]:='cartStatusWordIOJ2';
	gCSV_Buffer[3].aBuffer[Index[3]][c:=c+1]:=DINT_TO_STRING(i_safetyCheckVar.m_cartDriverInput[3].m_statusWord);  gCSV_Buffer[3].aBuffer[1][c]:='cartStatusWordIOJ3';
	gCSV_Buffer[3].aBuffer[Index[3]][c:=c+1]:=DINT_TO_STRING(i_safetyCheckVar.m_cartDriverInput[4].m_statusWord);  gCSV_Buffer[3].aBuffer[1][c]:='cartStatusWordIOJ4';
		
	//cart current joint motor encoder
	gCSV_Buffer[3].aBuffer[Index[3]][c:=c+1]:=DINT_TO_STRING(i_safetyCheckVar.m_cartDriverInput[1].m_motorEncoder);  gCSV_Buffer[3].aBuffer[1][c]:='cartCurMotorEncIOJ1';
	gCSV_Buffer[3].aBuffer[Index[3]][c:=c+1]:=DINT_TO_STRING(i_safetyCheckVar.m_cartDriverInput[2].m_motorEncoder);  gCSV_Buffer[3].aBuffer[1][c]:='cartCurMotorEncIOJ2';
	gCSV_Buffer[3].aBuffer[Index[3]][c:=c+1]:=DINT_TO_STRING(i_safetyCheckVar.m_cartDriverInput[3].m_motorEncoder);  gCSV_Buffer[3].aBuffer[1][c]:='cartCurMotorEncIOJ3';
	gCSV_Buffer[3].aBuffer[Index[3]][c:=c+1]:=DINT_TO_STRING(i_safetyCheckVar.m_cartDriverInput[4].m_motorEncoder);  gCSV_Buffer[3].aBuffer[1][c]:='cartCurMotorEncIOJ4';

	//cart commend joint motor encoder
	gCSV_Buffer[3].aBuffer[Index[3]][c:=c+1]:=DINT_TO_STRING(i_safetyCheckVar.m_cartDriverOutput[1].m_cmdMotorEncoder);  gCSV_Buffer[3].aBuffer[1][c]:='cartCmdMotorEncIOJ1';
	gCSV_Buffer[3].aBuffer[Index[3]][c:=c+1]:=DINT_TO_STRING(i_safetyCheckVar.m_cartDriverOutput[2].m_cmdMotorEncoder);  gCSV_Buffer[3].aBuffer[1][c]:='cartCmdMotorEncIOJ2';
	gCSV_Buffer[3].aBuffer[Index[3]][c:=c+1]:=DINT_TO_STRING(i_safetyCheckVar.m_cartDriverOutput[3].m_cmdMotorEncoder);  gCSV_Buffer[3].aBuffer[1][c]:='cartCmdMotorEncIOJ3';
	gCSV_Buffer[3].aBuffer[Index[3]][c:=c+1]:=DINT_TO_STRING(i_safetyCheckVar.m_cartDriverOutput[4].m_cmdMotorEncoder);  gCSV_Buffer[3].aBuffer[1][c]:='cartCmdMotorEncIOJ4';
	
	//output motor opMode IO
	gCSV_Buffer[3].aBuffer[Index[3]][c:=c+1]:=DINT_TO_STRING(i_safetyCheckVar.m_cartDriverOutput[1].m_opMode);  gCSV_Buffer[3].aBuffer[1][c]:='opModeIOJ1';
	gCSV_Buffer[3].aBuffer[Index[3]][c:=c+1]:=DINT_TO_STRING(i_safetyCheckVar.m_cartDriverOutput[2].m_opMode);  gCSV_Buffer[3].aBuffer[1][c]:='opModeIOJ2';
	gCSV_Buffer[3].aBuffer[Index[3]][c:=c+1]:=DINT_TO_STRING(i_safetyCheckVar.m_cartDriverOutput[3].m_opMode);  gCSV_Buffer[3].aBuffer[1][c]:='opModeIOJ3';
	gCSV_Buffer[3].aBuffer[Index[3]][c:=c+1]:=DINT_TO_STRING(i_safetyCheckVar.m_cartDriverOutput[4].m_opMode);  gCSV_Buffer[3].aBuffer[1][c]:='opModeIOJ4';
END_IF
END_METHOD

METHOD errCodeAnalysis : BOOL
VAR_INPUT
END_VAR

FOR i:=1 TO g_maxNum BY 1 DO
	IF g_ArrayErrCodeArm[i][0]<>0 AND ArrayErrCodeTypeLast[i]<> g_ArrayErrCodeArm[i][0]  THEN
		Arm:=SHR(g_ArrayErrCodeArm[i][0],24);
		IF Arm>g_maxNum THEN
			Arm:=g_maxNum;	
		END_IF
		Joint:=SHR(g_ArrayErrCodeArm[i][0],16) AND 16#FF;
		errID:=g_ArrayErrCodeArm[i][0];
		mErrNameLocation[arm,1]:=LREAL_TO_FMTSTR(arm,0, TRUE);
		mErrNameLocation[arm,2]:=LREAL_TO_FMTSTR(joint,0, TRUE);
		mErrNameLocation[arm,3]:=DWORD_TO_HEXSTR(UDINT_TO_DWORD(errID),0, TRUE);
		m_Index[arm]:=INT_TO_UDINT(Index[arm]);
		errWritingAllowed[arm]:=TRUE;
	END_IF
	ArrayErrCodeTypeLast[i]:=g_ArrayErrCodeArm[i][0];
	errFlagDelay1s[i](IN:= errWritingAllowed[i], PT:= T#2S, Q=> errWritingFalg[i], ET=> );
END_FOR
END_METHOD

METHOD run : BOOL
VAR_IN_OUT CONSTANT
	i_safetyCheckVar :ARRAY[1..g_maxNum] OF checkInputVariable;
	i_cartStatus : ST_CartStatus;
	i_cartJointData : ST_CartJointData;
	i_masterStatus :ST_MasterStatus;
	i_masterJointData : ST_MasterJointData;
END_VAR
_tNow := systemTime();
IF _tNow.wYear = 0 THEN
	RETURN;
END_IF

errCodeAnalysis();

armDataCast(i_safetyCheckVar,i_masterStatus,i_masterJointData);

cartDataCast(i_safetyCheckVar[g_cartNum],i_cartStatus,i_cartJointData);

FOR _iBuffer := 1 TO MAX_CSV_RING_BUFFER BY 1 DO
	TransferToWrittenVariable();

	WriterCSV();
	
	StartRecord[_iBuffer](CLK:=ErrWritingFalg[_iBuffer] , Q=> );

	IF ErrWritingFalg[_iBuffer] =FALSE THEN
		Index[_iBuffer]:=Index[_iBuffer]+1;
		IF Index[_iBuffer]>10000 THEN
			index[_iBuffer]:=2;
		END_IF
	END_IF
	
END_FOR
END_METHOD

METHOD systemTime : TIMESTRUCT
VAR_INPUT
END_VAR
fbSysTime(timeLoDW=>tFileTime.dwLowDateTime , timeHiDW=> tFileTime.dwHighDateTime);

_tNowBoLin := FILETIME_TO_SYSTEMTIME(tFileTime);
systemTime:=_tNowBoLin;
systemTime.wHour:=_tNowBoLin.wHour+8;
IF systemTime.wHour>23 THEN
	systemTime.wHour:=_tNow.wHour-24;
END_IF
END_METHOD

METHOD TransferToWrittenVariable : BOOL
VAR_INPUT
END_VAR

	gCSV_Buffer[_iBuffer].aBuffer[Index[_iBuffer]][0]:= SYSTEMTIME_TO_STRING(_tNow);(*第二行第一列*)
	gCSV_Buffer[_iBuffer].aBuffer[Index[_iBuffer]][1]:=LREAL_TO_FMTSTR(Index[_iBuffer],0, TRUE); 
	
	(*The first line shows the arm joint and the error name*)
	 mErrNameLocation[_iBuffer,0] := INT_TO_STRING(Index[_iBuffer]);
	gCSV_Buffer[_iBuffer].aBuffer[0][0] := mErrNameLocation[_iBuffer,0];
	gCSV_Buffer[_iBuffer].aBuffer[0][1] := mErrNameLocation[_iBuffer,1];
	gCSV_Buffer[_iBuffer].aBuffer[0][2] := mErrNameLocation[_iBuffer,2];
	gCSV_Buffer[_iBuffer].aBuffer[0][3] := mErrNameLocation[_iBuffer,3];
	//gCSV_Buffer[_iBuffer].aBuffer[4][0] := mErrNameLocation[_iBuffer,4];
	
	(*The second line shows the variable name*)
	gCSV_Buffer[_iBuffer].aBuffer[1][0] := 'SystemTime';
	gCSV_Buffer[_iBuffer].aBuffer[1][1] := 'Index';

	sPath:= 'C:\Robot\Error\'; 
	mErr[0]:=CONCAT('Arm',mErrNameLocation[_iBuffer,1]);
	mErr[1]:=CONCAT('Joint',mErrNameLocation[_iBuffer,2]);
	mErr[2]:=mErrNameLocation[_iBuffer,3];
	IF StartRecord[_iBuffer].Q THEN  
	gCSV_Buffer[_iBuffer].bFull := TRUE;
	fbFormat( 	sFormat := _sPathFormat ,
			 	arg1 := F_STRING(sPath),   arg2 := F_WORD(_tNow.wYear), arg3 := F_WORD(_tNow.wMonth), 
				arg4 := F_WORD(_tNow.wDay), arg5 := F_WORD(_tNow.wHour),arg6 := F_WORD(_tNow.wMinute),arg7 := F_WORD(_tNow.wSecond),
			    arg8 := F_STRING(mErr[0]),arg9 := F_STRING(mErr[1]),arg10 := F_STRING(mErr[2]),  sOut => gCSV_Buffer[_iBuffer].sPath);
	END_IF

	//F_STRING(mErr[0])
END_METHOD

METHOD writerCSV : BOOL
VAR_INPUT
END_VAR


	
	IF gCSV_Buffer[_iBuffer].bFull THEN

		gCSV_Buffer[_iBuffer].fbWriter(bWrite:= gCSV_Buffer[_iBuffer].bFull,sFileName:=gCSV_Buffer[_iBuffer].sPath, pBuffer :=ADR(gCSV_Buffer[_iBuffer].aBuffer),Index:=m_Index[_iBuffer]);
		gCSV_Buffer[_iBuffer].bFull := gCSV_Buffer[_iBuffer].fbWriter.bBusy;
	END_IF


	RecordCompletion[_iBuffer](CLK:= gCSV_Buffer[_iBuffer].bFull, Q=> );
	IF RecordCompletion[_iBuffer].Q THEN
		errWritingAllowed[_iBuffer]:=FALSE;
		Index[_iBuffer]:=2;
		gCSV_Buffer[_iBuffer].aBuffer:=iZeroRowsData;
		g_ArrayErrCodeArm[_iBuffer]:=iZeroErrCode[_iBuffer];
		//gCSV_Buffer[_iBuffer].fbWriter.arrDataForward(array_in:=Robot_Status.ArrayErrCodeType[_iBuffer]  , array_out=> Robot_Status.ArrayErrCodeType[_iBuffer]);
	END_IF
END_METHOD

END_FUNCTION_BLOCK

// ---- AgiMaths/MatrixLib/matTranspose.TcPOU
// B =A'
FUNCTION matTranspose : BOOL
VAR_IN_OUT CONSTANT
	matA :ARRAY[*,*] OF LREAL;
END_VAR

VAR_IN_OUT 
	matB :ARRAY[*,*] OF LREAL;
END_VAR

VAR
	i,j:DINT;
	m,n :DINT;
 
END_VAR

m:=UPPER_BOUND(matB,1);
n:= UPPER_BOUND(matB,2);
ASSERT(UPPER_BOUND(matA,1)=n);
ASSERT(UPPER_BOUND(matA,2)=m);
FOR i:=1 TO m DO
	FOR j:=1 TO n DO
		matB[i,j]:=matA[j,i];
	END_FOR
END_FOR

END_FUNCTION

// ---- AgiMaths/MatrixLib/matMultiply.TcPOU
// matC = matA * matB
FUNCTION matMultiply : BOOL
VAR_IN_OUT CONSTANT
	matA :ARRAY[*,*] OF LREAL;//m*p
	matB :ARRAY[*,*] OF LREAL;//p*n
END_VAR

VAR_IN_OUT 
	matC :ARRAY[*,*] OF LREAL;//m*n
END_VAR

VAR
	i,j, k :DINT;
	m,n,p :DINT;
	tmp:LREAL;
 
END_VAR

m:=UPPER_BOUND(matA,1);
p:=UPPER_BOUND(matA,2);
n:=UPPER_BOUND(matB,2);
ASSERT(UPPER_BOUND(matB,1)=p);
ASSERT(UPPER_BOUND(matC,1)=m);
ASSERT(UPPER_BOUND(matC,2)=n);

FOR i:=1 TO m DO
	FOR j:=1 TO n DO
		matC[i,j]:=0.0;
	END_FOR
END_FOR

FOR i:=1 TO m DO
	FOR k:=1 TO p DO
		tmp:=matA[i,k];
		FOR j:=1 TO n DO 
		matC[i,j]:=matC[i,j]+tmp*matB[k,j];
		END_FOR
	END_FOR
END_FOR

END_FUNCTION

// ---- AgiMaths/MatrixLib/rot2AngAxis.TcPOU
FUNCTION rot2AngAxis : bool
VAR_IN_OUT CONSTANT
	rot : Mat3d;
END_VAR
VAR_OUTPUT
	angle: LREAL;
	axis : Vec3d;
END_VAR
VAR
	tmp:LREAL;
END_VAR

tmp:=LIMIT(-1, (rot[1,1]+rot[2,2]+rot[3,3]-1)/2 , 1);
angle := ACOS(tmp);

// no rotation
IF ABS(angle)<g_smallAng THEN
	angle :=0;
	axis[1]:=1;
	axis[2]:=0;
	axis[3]:=0;
// rotate pi
ELSIF ABS(angle-pi)< g_smallAng THEN
	angle :=PI;
	axis[1]:=SQRT((rot[1,1]+1)/2);
	axis[2]:=SQRT((rot[2,2]+1)/2);
	axis[3]:=SQRT((rot[3,3]+1)/2);
	IF axis[1]>g_smallNum THEN
		axis[2]:=0.5*rot[1,2]/axis[1];
		axis[3]:=0.5*rot[1,3]/axis[1];
	ELSIF axis[2]>g_smallNum THEN
		axis[1]:=0.5*rot[2,1]/axis[2];
		axis[3]:=0.5*rot[2,3]/axis[2];
	ELSE
		axis[1]:=0.5*rot[3,1]/axis[3];
		axis[2]:=0.5*rot[3,2]/axis[3];
	END_IF
// others
ELSE
	tmp:=2*SIN(angle);
	axis[1]:=(rot[3,2]-rot[2,3])/tmp;
	axis[2]:=(rot[1,3]-rot[3,1])/tmp;
	axis[3]:=(rot[2,1]-rot[1,2])/tmp;
END_IF

// normalize
normalize(axis);

END_FUNCTION

// ---- AgiMaths/MatrixLib/normalize.TcPOU
// normalize the input vector
FUNCTION normalize : BOOL
VAR_IN_OUT
	vec :ARRAY[*] OF LREAL;
END_VAR
VAR
	m,i:DINT;
	vecNorm :LREAL;
END_VAR

m:=UPPER_BOUND(vec,1);
vecNorm :=norm(vec);

// if vector close to zero, remain the same;
IF vecNorm< g_smallNum THEN
	normalize :=FALSE;
	RETURN;
END_IF

FOR i:=1 TO m DO
	vec[i] := vec[i]/vecNorm;
END_FOR
normalize :=TRUE;

END_FUNCTION

// ---- AgiMaths/MatrixLib/norm.TcPOU
// return the norm of a vector
FUNCTION norm : LREAL
VAR_IN_OUT CONSTANT
	vec :ARRAY[*] OF LREAL;
END_VAR
VAR
	m,i:DINT;
END_VAR

m:=UPPER_BOUND(vec,1);
norm:=0;
FOR i:=1 TO m DO
	norm := norm + vec[i]*vec[i];
END_FOR

norm := SQRT(norm);

END_FUNCTION

// ---- AgiMaths/MatrixLib/vecMultiNum.TcPOU
// vecB=VecA*num
FUNCTION vecMultiNum : BOOL
VAR_IN_OUT CONSTANT
	vecA :ARRAY[*] OF LREAL;
END_VAR

VAR_INPUT
	num :LREAL;
END_VAR

VAR_IN_OUT
	vecB : ARRAY[*] OF LREAL;
END_VAR
VAR
	m :DINT;
	i :DINT;
END_VAR

m:=UPPER_BOUND(vecA,1);
ASSERT(UPPER_BOUND(VecB,1)=m);

FOR i:=1 TO m DO
		vecB[i]:=num*vecA[i];
END_FOR

END_FUNCTION

// ---- SafetyCheck/FB_EtherCATCheck.TcPOU
FUNCTION_BLOCK FB_EtherCATCheck
VAR_INPUT
END_VAR
VAR_OUTPUT
END_VAR
VAR
	//drive EtherCAT communition detection
	m_commuEtherCATState:FB_EcGetSlaveState;
	m_EcSlaveState : ST_EcSlaveState;
	
	m_crcVerify : FB_EcGetSlaveCrcError;
	m_crcError : ST_EcCrcError;
	
	m_EtherCATVerify : ST_EtherCATState;
END_VAR

METHOD EtherCATVerify : ST_EtherCATState
VAR_INPUT
	armsNetID:T_AmsNetID;
	jntAddr:UINT;
END_VAR

m_commuEtherCATState(sNetId:= armsNetID, nSlaveAddr:= jntAddr, bExecute:= TRUE, tTimeout:= , bBusy=> , bError=> , nErrId=> , state=> m_EcSlaveState);

IF NOT m_commuEtherCATState.bBusy THEN
	m_commuEtherCATState(bExecute:=FALSE);
	IF m_EcSlaveState.deviceState = EC_DEVICE_STATE_OP THEN
		m_EtherCATVerify.EtherCATState := TRUE;
	ELSE
		m_EtherCATVerify.EtherCATState := FALSE;
	END_IF
END_IF


m_crcVerify(sNetId:= armsNetID, nSlaveAddr:= jntAddr, bExecute:= TRUE, tTimeout:= , bBusy=> , bError=> , nErrId=> , crcError=> m_crcError);
IF NOT m_crcVerify.bBusy THEN
	m_crcVerify(bExecute:=FALSE);
	m_EtherCATVerify.CRCPortA := MAX(EtherCATVerify.CRCPortA,m_crcError.portA);
	m_EtherCATVerify.CRCPortB := MAX(EtherCATVerify.CRCPortB,m_crcError.portB);
	m_EtherCATVerify.CRCPortC := MAX(EtherCATVerify.CRCPortC,m_crcError.portC);
END_IF

EtherCATVerify := m_EtherCATVerify;
END_METHOD

END_FUNCTION_BLOCK

// ---- Mains/CartControl.TcPOU
PROGRAM CartControl
VAR
	// cart instance
	m_masterCart :FB_MasterCart;
	
	//cart related UI
	m_cartUIData : ST_CartUIData;
	
	// Output cart status
	m_cartStatus AT%Q* : ST_CartStatus;
	
	// Cart  joint data
	m_cartJointData AT %Q* :ST_CartJointData;
	
	// wait time before cart init for ethercat to be statble 
	m_cartInitWaitTime : LREAL:=0;
	
	// cart init flag
	m_cartInit :BOOL :=FALSE;
	
	m_workHeartTon0 : TON;
	m_workHeartTon1 : TON;
	m_ergonInfoHeightF : F_TRIG;
	m_userLoggedR : R_TRIG;
	m_ergonInfoHeight : BOOL;
END_VAR

// wait communication to be stable
IF(m_cartInitWaitTime<g_robotInitWaitTime) THEN
	m_cartInitWaitTime := m_cartInitWaitTime+g_armCtrlCycleTime;
	RETURN;
END_IF

// cart init
IF m_cartInit =FALSE THEN
	m_masterCart.Init();
	m_cartInit:=TRUE;
END_IF

// input from UI
UIInputProcess();

// cart run
m_masterCart.run(m_cartUIData);

// status/joint data output
m_masterCart.getStatus(m_cartStatus, m_cartJointData);

// tranform data from UI(global variable write by ADS) to ST_UIData
METHOD UIInputProcess : BOOL
VAR_INPUT
END_VAR
//init cart joint postion
IF (GVL_interactUI.g_uiParaReload=TRUE) THEN
	GVL_interactUI.g_uiParaReload:=FALSE;
	m_cartUIData.m_cmdCancelErgonPos := m_cartJointData.m_curJntPos;
	m_cartUIData.m_cmdJntPos:= g_zeroVec4d;
	GVL_interactUI.g_ergonomicCtrl.m_ergonInfoModify:=TRUE;
END_IF

//recover the ergonomic button and cancel recover ergonomic button
m_cartUIData.m_ergonomicCrl.m_recovErgonEnable := GVL_interactUI.g_ergonomicCtrl.m_recovErgonEnable;
m_cartUIData.m_ergonomicCrl.m_cancelRecovErgonEnable := GVL_interactUI.g_ergonomicCtrl.m_cancelRecovErgonEnable;

//recover the ergonomic update commend position
m_userLoggedR(CLK:= GVL_interactUI.g_userLogged, Q=> );
IF m_userLoggedR.Q THEN
	m_cartUIData.m_cmdJntPos:= g_zeroVec4d;
END_IF
IF ((GVL_interactUI.g_ergonomicCtrl.m_recovErgonEnable AND NOT GVL_interactUI.g_ergonomicCtrlEnableLast.m_recovErgonEnable))  THEN
	GVL_interactUI.g_ergonomicCtrl.m_recovErgonFinshed:=FALSE;
	m_cartUIData.m_cmdCancelErgonPos := m_cartJointData.m_curJntPos;
	m_cartUIData.m_cmdJntPos[1] := GVL_interactUI.g_ergonomicCtrlData.m_monitorHeight;
	m_cartUIData.m_cmdJntPos[2] := GVL_interactUI.g_ergonomicCtrlData.m_headAngle;
	m_cartUIData.m_cmdJntPos[3] := GVL_interactUI.g_ergonomicCtrlData.m_handrailHeight;
	m_cartUIData.m_cmdJntPos[4] := GVL_interactUI.g_ergonomicCtrlData.m_footDistance;
END_IF

//cancel recover the ergonomic update commend position
IF (GVL_interactUI.g_ergonomicCtrlEnableLast.m_cancelRecovErgonEnable=FALSE) AND (GVL_interactUI.g_ergonomicCtrl.m_cancelRecovErgonEnable=TRUE) THEN
	GVL_interactUI.g_ergonomicCtrl.m_cancelRecovErgonFinshed:=FALSE;
	m_cartUIData.m_cmdJntPos := m_cartUIData.m_cmdCancelErgonPos;
END_IF
GVL_interactUI.g_ergonomicCtrlEnableLast:=GVL_interactUI.g_ergonomicCtrl;

GVL_interactUI.g_ergonomicCtrl.m_cancelRecovErgonFinshed := m_cartStatus.m_cancelErgonAdjustArrival;
GVL_interactUI.g_ergonomicCtrl.m_recovErgonFinshed := m_cartStatus.m_ergonAdjustArrival;
GVL_interactUI.g_surgonHeadIn:=m_cartStatus.m_surgonReady;

//cart adjustment complete , update ui information
m_ergonInfoHeightF(CLK:= m_cartStatus.m_consoleInAdjust, Q=>m_ergonInfoHeight);
IF m_ergonInfoHeight THEN
	GVL_interactUI.g_ergonomicCtrl.m_ergonInfoModify := TRUE;
END_IF
GVL_interactUI.g_ergonomicCurData.m_monitorHeight := m_cartJointData.m_curJntPos[1];
GVL_interactUI.g_ergonomicCurData.m_headAngle := m_cartJointData.m_curJntPos[2];
GVL_interactUI.g_ergonomicCurData.m_handrailHeight := m_cartJointData.m_curJntPos[3];
GVL_interactUI.g_ergonomicCurData.m_footDistance:= m_cartJointData.m_curJntPos[4];
GVL_interactUI.g_cartInMotion := m_cartStatus.m_consoleInManualAdjust;


//work heart
m_workHeartTon0(IN:= GVL_interactUI.g_heartBeat = 1, PT:= T#1S, Q=> , ET=> );
m_workHeartTon1(IN:= GVL_interactUI.g_heartBeat = 0, PT:= T#1S, Q=> , ET=> );
IF m_workHeartTon0.Q THEN
	GVL_interactUI.g_heartBeat :=0 ;
ELSIF m_workHeartTon1.Q THEN
	GVL_interactUI.g_heartBeat  :=1 ;
END_IF
END_METHOD

END_PROGRAM

// ---- FBs_Robots/FB_MasterCart.TcPOU
FUNCTION_BLOCK FB_MasterCart
VAR
	//  IO and check
	m_endoScopePedalIO AT%I* :BOOL;
	m_endoScopeIOCheck :FB_IOCheck;
	
	m_clutchPedalIO AT%I* :BOOL;
	m_clutchIOCheck :FB_IOCheck;
	
	m_surgonHeadInIO AT%I* :BOOL;
	m_headInCheck:FB_IOCheck;
	
	m_armSwitchIO AT%I* :BOOL;
	m_armSwitchCheck:FB_IOToggleCheck;
	
	m_electricCutLeft AT %I* :BOOL;
	m_electricCutLeftAllow AT %I* :BOOL;
	
	m_electricCutRight AT %I* :BOOL;
	m_electricCutRightAllow AT %I* :BOOL;
	
	m_electricCoagulLeft AT %I* :BOOL;
	m_electricCoagulLeftAllow AT %I* :BOOL;
	
	m_electricCoagulRight AT %I* :BOOL;
	m_electricCoagulRightAllow AT %I* :BOOL;
	
	m_elecKnifeCtrlWord AT %Q* :DINT;
	
	// cart status
	m_cartStatus  : ST_CartStatus;
	
	// cart joints
	// [monitor lift, monitor rotate, armset, pedal]
	m_cartJoints:ARRAY[1..4] OF FB_CartJoint;
	
	// cart joint motion control IO
	//[monitor_up, monitor_down, monitor_cwRotate, monitor_ccwRotate, armset_up, armset_down, pedal_in, pedal_out]
	m_cartJointCtrlIO AT%I* :ARRAY[1..8] OF BOOL ;
	m_cartJointCtrlIOCheck :ARRAY[1..8] OF FB_IOCheck;
	
	//electrotome control io
	m_electricCutLeftOn :BOOL;
	m_electricCutRightOn :BOOL;
	m_electricCoagulLeftOn : BOOL;
	m_electricCoagulRightOn : BOOL;
	//Triggering several energies at once
	m_eleCtrlState : UINT;
	//The type of instrument energy of the master hand corresponding to the slave hand
	m_energyType :ARRAY[1..g_mArmNum] OF UINT :=[2(0)];
	
	// cart joint control data
	m_jntEnableCounts:Vec4i ;
	m_jntDisableCounts:Vec4i ;
	m_jntEnableCountsThres:INT:=500;
	m_jntCmdMotionDir :Vec4i;
	m_cmdJntTrq :Vec4d;
	m_cmdJntPos :Vec4d;
	m_cmdJntVel :Vec4d;
	m_jntEnableFlag :Vec4b;
	
	//cart ergonomic adjust data
	m_UIData : ST_CartUIData;
	m_carInMotion : INT; // 0:  no mition, 1: mamual adjust, 2: ergonomic adjust
	m_jntSoftwareLimit :ARRAY [1..4] OF LREAL := [0.001, 1*g_deg2Rad, 0.001, 0.001];
	m_cmdArrival : Vec4b;
	
	// cart joint status data
	m_curMotorPos :Vec4d;
	m_curLinkPos :Vec4d;
	m_curJntPos :Vec4d;
	m_curJntVel :Vec4d;
	m_curJntTrq :Vec4d;
	m_rawJntCurrent :Vec4d;
	m_filtJntCurrent :Vec4d;
	m_cmdJntCurrent : Vec4d;

END_VAR

METHOD eleKnifeCtrl : DINT
VAR_IN_OUT CONSTANT
	m_armState:ARRAY[1..g_mArmNum] OF E_masterArmState ;
	m_teleSlaveArmIdx :ARRAY[1..g_mArmNum] OF E_MatchedSlaveArmIdx;
	m_instruStauts: ARRAY[1..g_sArmNum] OF ST_InstruStatus;
END_VAR

//Foot trigger check
m_electricCutLeftOn := m_electricCutLeft AND m_electricCutLeftAllow AND m_armState[1] = MasterArmState_MasterSlave ;
m_electricCutRightOn := m_electricCutRight AND m_electricCutRightAllow AND m_armState[2] = MasterArmState_MasterSlave ;
m_electricCoagulLeftOn := m_electricCoagulLeft AND m_electricCoagulLeftAllow AND m_armState[1] = MasterArmState_MasterSlave ;
m_electricCoagulRightOn := m_electricCoagulRight AND m_electricCoagulRightAllow AND m_armState[2] = MasterArmState_MasterSlave ;

//You cannot excite two energies at the same time
m_eleCtrlState := BOOL_TO_UINT(m_electricCutLeftOn) + BOOL_TO_UINT(m_electricCutRightOn)
										 + BOOL_TO_UINT(m_electricCoagulLeftOn) + BOOL_TO_UINT(m_electricCoagulRightOn);

IF m_teleSlaveArmIdx[1] > 0 THEN
	m_energyType[1] := m_instruStauts[m_teleSlaveArmIdx[1]].m_energyType;
	m_energyType[2] := m_instruStauts[m_teleSlaveArmIdx[2]].m_energyType;
END_IF

IF m_eleCtrlState = 1 THEN
	IF (m_electricCutLeftOn AND  m_energyType[1] = InstruType_isMonopole) OR (m_electricCutRightOn AND  m_energyType[2] = InstruType_isMonopole) THEN
		eleKnifeCtrl := EnergyCtrlWord_isMonopoleCut;
	ELSIF (m_electricCoagulLeftOn AND m_energyType[1] = InstruType_isMonopole) OR (m_electricCoagulRightOn AND  m_energyType[2] = InstruType_isMonopole) THEN
		eleKnifeCtrl := EnergyCtrlWord_isMonopoleCoagul;
	ELSIF (m_electricCoagulLeftOn AND m_energyType[1] = InstruType_isBipolar) OR (m_electricCoagulRightOn AND  m_energyType[2] = InstruType_isBipolar) THEN
		eleKnifeCtrl := EnergyCtrlWord_isBipolarCoagul;
	ELSIF (m_electricCutLeftOn AND m_energyType[1] = InstruType_isUltraKnife) OR (m_electricCutRightOn AND  m_energyType[2] = InstruType_isUltraKnife) THEN
		eleKnifeCtrl := EnergyCtrlWord_isUltraMin;
	ELSIF (m_electricCoagulLeftOn AND m_energyType[1] = InstruType_isUltraKnife) OR (m_electricCoagulRightOn AND  m_energyType[2] = InstruType_isUltraKnife) THEN
		eleKnifeCtrl := EnergyCtrlWord_isUltraMax;
		
	ELSE
		eleKnifeCtrl := EnergyCtrlWord_NoOutput;
	END_IF
ELSE
	eleKnifeCtrl := EnergyCtrlWord_NoOutput;
END_IF
END_METHOD

METHOD ergonomicAdjust : INT
VAR_INPUT
END_VAR
VAR
	i : INT;
	err:Vec4d;
END_VAR
vecSub(m_UIData.m_cmdJntPos,m_curJntPos, err);
ergonomicAdjust := 2;
//only update command after joints is truly enabled
FOR i := 1 TO 4 DO
	IF m_jntEnableFlag[i] AND m_cartJoints[i].isEnabled() AND m_jntEnableCounts[i]>= m_jntEnableCountsThres THEN
		m_cmdJntVel[i]:=sign(m_UIData.m_cmdJntPos[i]-m_cartJoints[i].jntPos)*(GVL_CartJointParameters.g_jntCtrlMotionVel[i]);
		IF ABS(err[i]) < m_jntSoftwareLimit[i]/3 THEN
			m_cmdJntVel[i]:=0;
		END_IF
		m_cmdJntPos[i] := LIMIT(GVL_CartJointParameters.g_minJntPos[i] + m_jntSoftwareLimit[i],  m_cmdJntPos[i] + m_cmdJntVel[i]*g_cartCtrlCycleTime, GVL_CartJointParameters.g_maxJntPos[i] - m_jntSoftwareLimit[i]);
	
	ELSE
		m_cmdJntVel[i]:=0;
		m_cmdJntPos[i] := m_cartJoints[i].jntPos;
	END_IF	
END_FOR
END_METHOD

METHOD PUBLIC getStatus : BOOL
VAR_IN_OUT
	// cart status data
	r_cartStatus :ST_CartStatus;
	
	// cart joint data
	r_cartJointData :ST_CartJointData;
	
END_VAR
r_cartStatus := m_cartStatus;


// current joint data
r_cartJointData.m_curMotorPos:=m_curMotorPos;
r_cartJointData.m_curLinkPos:=m_curLinkPos;
r_cartJointData.m_curJntPos:=m_curJntPos;
r_cartJointData.m_curJntVel:=m_curJntVel;
r_cartJointData.m_curJntTrq:=m_curJntVel;
r_cartJointData.m_rawJntCurrent:=m_rawJntCurrent;
r_cartJointData.m_filtJntCurrent:=m_filtJntCurrent;

// command joint data
r_cartJointData.m_cmdJntPos:=m_cmdJntPos;
r_cartJointData.m_cmdJntVel:=m_cmdJntVel;
r_cartJointData.m_cmdJntTrq:=m_cmdJntTrq;
r_cartJointData.m_cmdJntCurrent:=m_cmdJntCurrent;
END_METHOD

METHOD PUBLIC init : BOOL
VAR_INPUT
END_VAR
VAR
	i:INT;
	initLinkPos :LREAl;
END_VAR
// joint init
FOR i:=1 TO 4 DO
	m_cartJoints[i].init(i,g_cartCtrlCycleTime);
	m_cartJoints[i].initJntPos();
END_FOR

// motor and link encoder of  monitor rotation are on different  joints
// transfer monitor angle from link side to motor side
initLinkPos:= monitorAngLink2Motor(m_cartJoints[2].initLinkPos);
m_cartJoints[2].initJntPosReset(initLinkPos);

// init commands
FOR i:=1 TO 4 DO
	m_jntEnableCounts[i]:=0;
	m_jntDisableCounts[i]:=0;
	m_jntEnableFlag[i]:=FALSE;
	m_jntCmdMotionDir[i]:=0;
	m_cmdJntTrq[i]:=0;
	m_cmdJntVel[i]:=0;
	m_cmdJntPos[i]:=m_cartJoints[i].jntPos;
END_FOR

m_cartStatus.m_initFlag :=true;
END_METHOD

METHOD manualAdjust : INT
VAR_INPUT
END_VAR
VAR
	i : INT;
END_VAR
// update joint command positon
manualAdjust := 1;
//only update command after joints is truly enabled
FOR i := 1 TO 4 DO
	IF  m_jntEnableFlag[i] AND m_cartJoints[i].isEnabled() AND m_jntEnableCounts[i]>= m_jntEnableCountsThres THEN
		//  update command joint velocity
		m_cmdJntVel[i]:=m_jntCmdMotionDir[i]*GVL_CartJointParameters.g_jntCtrlMotionVel[i];
		
		// limit handle
		IF (m_cmdJntPos[i]> GVL_CartJointParameters.g_maxJntPos[i] AND m_cmdJntVel[i] >0 ) OR 
				(m_cmdJntPos[i]< GVL_CartJointParameters.g_minJntPos[i] AND m_cmdJntVel[i] <0 )  THEN
				m_cmdJntVel[i] := 0.0;
		END_IF
		m_cmdJntPos[i]:= m_cmdJntPos[i]+ m_cmdJntVel[i]*g_cartCtrlCycleTime;
	ELSE
		m_cmdJntVel[i]:=0;
		m_cmdJntPos[i] := m_cartJoints[i].jntPos;
	END_IF
END_FOR
END_METHOD

// TODO
METHOD PROTECTED monitorAngLink2Motor : LREAL
VAR_INPUT
	i_linkPos:LREAL;
END_VAR
VAR
	A,B,C,D,E,F,G,H,I,X0,X1,X2,X3,X4,X5,X6,X7,X8,X9,X10,X11,X12,Z0:LREAL;	
	offset :LREAL := 0.8877;
END_VAR

X0:=i_linkPos+offset;  //监视器旋转

A:=227; B:=216; C:=159.285; D:=150.297; E:=195; F:=130; G:=137; H:=40; I:=99;
X4:=ATAN(H/I); X5:=ATAN(F/G);
X8:=SQRT(F*F+G*G);
X12:=sqrt(H*H+I*I);
X9:=sqrt(E*E+X12*X12-2*E*X12*cos(X0));
X6:=acos((B*B+X8*X8-X9*X9)/(2*B*X8));
X10:=acos((B*B+X9*X9-X8*X8)/(2*B*X9));
X11:=acos((X9*X9+X12*X12-E*E)/(2*X9*X12));
X7:=X10+X11;
X2:=X5-X6;
X3:=pi-X7+X2;
X1:=X3-X4;

monitorAngLink2Motor:=-X2;
END_METHOD

//TODO
METHOD PROTECTED monitorAngMotor2Link : LREAL
VAR_INPUT
	i_motorPos:LREAL;
END_VAR
VAR
	A,B,C,D,E,F,G,H,I,X0,X1,X2,X3,X4,X5,X6,X7,X8,X9,X10,X11,X12,Z0:LREAL;	
	offset :LREAL := 0.8877;
END_VAR
X2:=-i_motorPos;

A:=227; B:=216; C:=159.285; D:=150.297; E:=195; F:=130; G:=137; H:=40; I:=99;
X5:=atan(F/G);
X6:=X5-X2;
X8:=sqrt(F*F+G*G);
X9:=sqrt(B*B+X8*X8-2*B*X8*cos(X6));
X12:=SQRT(H*H+I*I);
X0:=ACOS((E*E+X12*X12-X9*X9)/(2*E*X12));

monitorAngMotor2Link:=X0-offset;
END_METHOD

METHOD reachUITargetCheck : bool
VAR
	i :INT;
	err:Vec4d;
END_VAR
vecSub(m_UIData.m_cmdJntPos,m_curJntPos, err);

// joint error check
FOR i:=1 TO 4 DO 
	m_cmdArrival[i] :=  ABS(err[i]) < m_jntSoftwareLimit[i]/2;
END_FOR
END_METHOD

METHOD PUBLIC run : BOOL
VAR_IN_OUT CONSTANT
	i_cartUIData : ST_CartUIData;
END_VAR
VAR
	i:INT;
END_VAR
// update IO signals
updateIO(i_cartUIData);

// update cart status
updateStatus();

// update controller and command
updateCmds();

// send command to joint driver
FOR i:=1 TO 4 DO
	// joint enable
	IF m_jntEnableFlag[i] AND NOT(SafetyCheck.m_safetyCheckData.m_cartErrFlag[i]) AND MasterArmControl.m_masterStatus.m_armState[1] <> MasterArmState_MasterSlave 
								AND MasterArmControl.m_masterStatus.m_armState[2] <> MasterArmState_MasterSlave THEN
		m_cartJoints[i].enable();
	ELSE
		m_cartJoints[i].disable();
	END_IF
	
	// set command position
	m_cartJoints[i].updateCmds(DriverOPMode_Pos,m_cmdJntPos[i],m_cmdJntTrq[i]);
END_FOR
END_METHOD

PROPERTY status : ST_CartStatus
GET
status := m_cartStatus;
END_GET
END_PROPERTY

METHOD PROTECTED updateCmds : BOOL
VAR_INPUT
END_VAR
VAR
	i:INT;
	
END_VAR
IF (m_jntCmdMotionDir[1] <>0 OR m_jntCmdMotionDir[2]<>0 OR m_jntCmdMotionDir[3] <>0 OR m_jntCmdMotionDir[4] <>0) AND m_carInMotion <> 2 THEN
	m_carInMotion := manualAdjust();
ELSIF (m_UIData.m_ergonomicCrl.m_recovErgonEnable OR m_UIData.m_ergonomicCrl.m_cancelRecovErgonEnable) AND m_carInMotion <> 1 THEN
	m_carInMotion := ergonomicAdjust();
ELSE
	m_carInMotion := 0;
END_IF

reachUITargetCheck();
IF m_cmdArrival[1] AND m_cmdArrival[2] AND m_cmdArrival[3] AND m_cmdArrival[4] THEN
	IF m_UIData.m_ergonomicCrl.m_recovErgonEnable THEN
		m_cartStatus.m_cancelErgonAdjustArrival := FALSE;
		m_cartStatus.m_ergonAdjustArrival := TRUE;
	END_IF
	IF m_UIData.m_ergonomicCrl.m_cancelRecovErgonEnable THEN
		m_cartStatus.m_ergonAdjustArrival := FALSE;
		m_cartStatus.m_cancelErgonAdjustArrival := TRUE;
	END_IF
ELSE
	m_cartStatus.m_ergonAdjustArrival := FALSE;
	IF m_UIData.m_ergonomicCrl.m_recovErgonEnable THEN
		m_cartStatus.m_cancelErgonAdjustArrival := FALSE;
	END_IF
END_IF
END_METHOD

METHOD PROTECTED updateIO : BOOL
VAR_INPUT
	i_cartUIData : ST_CartUIData;
END_VAR
VAR
	i:INT;
	idxOffset:INT;
END_VAR
// updata IO signals
m_cartStatus.m_clutchSwitch:= m_clutchIOCheck.check(m_clutchPedalIO);
m_cartStatus.m_endoscopeSwitch := m_endoScopeIOCheck.check(m_endoScopePedalIO);
m_cartStatus.m_surgonReady := m_headInCheck.check(m_surgonHeadInIO);
m_cartStatus.m_armSwitch :=m_armSwitchCheck.check(m_armSwitchIO);
m_UIData := i_cartUIData;

//updata Electrotome control
m_elecKnifeCtrlWord := eleKnifeCtrl(MasterArmControl.m_masterStatus.m_armState , MasterArmControl.m_masterStatus.m_teleSlaveArmIdx , MasterArmControl.m_masterInputDataPool.m_slaveStatus.m_instruStauts );

//updata pedal hover and pedal trigger
m_cartStatus. m_pedalHover[1] := m_electricCutLeftAllow OR m_electricCoagulLeftAllow;
m_cartStatus. m_pedalHover[2] := m_electricCutRightAllow OR m_electricCoagulRightAllow;
IF m_electricCutLeftOn AND m_eleCtrlState = 1 THEN
	m_cartStatus.m_electricKnifePedalTrigger[1] := 1;
ELSIF m_electricCoagulLeftOn AND m_eleCtrlState = 1 THEN
	m_cartStatus.m_electricKnifePedalTrigger[1] := 2;
ELSE
	m_cartStatus.m_electricKnifePedalTrigger[1] := 0;
END_IF

IF m_electricCutRightOn AND m_eleCtrlState = 1 THEN
	m_cartStatus.m_electricKnifePedalTrigger[2] := 1;
ELSIF m_electricCoagulRightOn AND m_eleCtrlState = 1 THEN
	m_cartStatus.m_electricKnifePedalTrigger[2] := 2;
ELSE
	m_cartStatus.m_electricKnifePedalTrigger[2] := 0;
END_IF

//update cart joint control switch
FOR i:=1 TO 4 DO 
	idxOffset:= 2*(i-1);
	IF m_cartJointCtrlIOCheck[1+idxOffset].check(m_cartJointCtrlIO[1+idxOffset]) THEN
		m_jntCmdMotionDir[i]:=1;
	ELSIF  m_cartJointCtrlIOCheck[2+idxOffset].check(m_cartJointCtrlIO[2+idxOffset]) THEN
		m_jntCmdMotionDir[i]:=-1;
	ELSE
		m_jntCmdMotionDir[i]:=0;
	END_IF
END_FOR


// if console is already in motion, only check the currently moving joint
IF m_cartStatus.m_consoleInAdjust THEN
	FOR i:=1 TO 4 DO
		IF NOT(m_cartJoints[i].isEnabled()) THEN
			m_jntCmdMotionDir[i] := 0;
		END_IF
	END_FOR
END_IF


// update joint enable flag
FOR i:= 1 TO 4 DO
	IF m_jntCmdMotionDir[i] <> 0 OR m_UIData.m_ergonomicCrl.m_recovErgonEnable OR m_UIData.m_ergonomicCrl.m_cancelRecovErgonEnable THEN
		m_jntEnableFlag[i] := TRUE;
		m_jntEnableCounts[i]:= LIMIT(0, m_jntEnableCounts[i]+1, m_jntEnableCountsThres);
		m_jntDisableCounts[i]:=m_jntEnableCountsThres;
	ELSE
		m_jntEnableCounts[i]:=0;
		m_jntDisableCounts[i]:= LIMIT(0, m_jntDisableCounts[i]-1, m_jntEnableCountsThres);
		m_jntEnableFlag[i] :=m_jntDisableCounts[i]>0; 
	END_IF
END_FOR


// Do not adjust during master-slave control
IF MasterArmControl.m_masterStatus.m_armState[1] = MasterArmState_MasterSlave OR MasterArmControl.m_masterStatus.m_armState[1] = MasterArmState_Endoscope OR
	MasterArmControl.m_masterStatus.m_armState[2] = MasterArmState_MasterSlave OR MasterArmControl.m_masterStatus.m_armState[2] = MasterArmState_Endoscope  THEN
	m_jntCmdMotionDir := g_zeroVec4i;
END_IF
END_METHOD

METHOD PROTECTED updateStatus : BOOL
VAR_INPUT
END_VAR
VAR
	i:INT;
END_VAR
// update cart joints status
FOR i:=1  TO 4 DO
	m_cartJoints[i].updateStatus();
END_FOR

// get joint data
FOR i:=1 TO 4 DO
	m_curMotorPos[i]:=m_cartJoints[i].motorPos;
	m_curLinkPos[i]:=m_cartJoints[i].linkPos;
	m_curJntPos[i]:=m_cartJoints[i].jntPos;
	m_curJntVel[i]:=m_cartJoints[i].jntVel;
	m_curJntTrq[i]:=m_cartJoints[i].jntTrq;
	m_rawJntCurrent[i]:=m_cartJoints[i].rawCurrent;
	m_filtJntCurrent[i]:=m_cartJoints[i].filtCurrent;
	m_cmdJntCurrent[i]:=m_cartJoints[i].cmdCurrent;
END_FOR 

// transfer monitor angle from link side to motor side
m_curLinkPos[2]:= monitorAngLink2Motor(m_curLinkPos[2]);

// get monitor angle
m_cartStatus.m_monitorAngle:= m_cartJoints[2].linkPos;

// check if cart in motion
m_cartStatus.m_consoleInAdjust:=FALSE;
FOR i:=1 TO 4 DO
	IF m_cartJoints[i].isEnabled() THEN
		m_cartStatus.m_consoleInAdjust:=TRUE;
		EXIT;
	END_IF
END_FOR
// check if cart in manual adjustment
m_cartStatus.m_consoleInManualAdjust := FALSE;
FOR i:=1 TO 4 DO
	IF m_jntCmdMotionDir[i] <> 0 AND m_cartJoints[i].isEnabled() THEN
		m_cartStatus.m_consoleInManualAdjust := TRUE;
		EXIT;
	END_IF
END_FOR
END_METHOD

END_FUNCTION_BLOCK

// ---- FBs_Auxiliary/FB_IOCheck.TcPOU
FUNCTION_BLOCK FB_IOCheck
VAR
	// IO type, 0- normally-opend IO; 1- normally-closed IO
	m_IOType :INT :=0;
	
	// counts after IO  is triggerd
	m_IOOnCounts :INT;
	
	// counts threshold indicating IO is trully triggerd
	m_IOOnCountThres :INT :=100;
END_VAR

METHOD check : BOOL
VAR_INPUT
	IOValue :BOOL;
END_VAR
IF (0=m_IOType and IOValue) OR (1=m_IOType AND NOT(IOValue)) THEN
	m_IOOnCounts := MIN(m_IOOnCounts +1, m_IOOnCountThres);
ELSE
	 m_IOOnCounts :=0;
END_IF

check:=m_IOOnCounts>=m_IOOnCountThres;
END_METHOD

METHOD init : BOOL
VAR_INPUT
	i_IOType :INT;
	i_triggerCounts:INT;
END_VAR
m_IOType:=i_IOType;
m_IOOnCountThres := i_triggerCounts;
END_METHOD

END_FUNCTION_BLOCK

// ---- FBs_Auxiliary/FB_IOToggleCheck.TcPOU
// return true if IO is triggerd for a set time period
// only return ture for one cycle, waiting for IO to be released and check for next time
FUNCTION_BLOCK FB_IOToggleCheck
VAR
	// IO type, 0- normally-opend IO; 1- normally-closed IO
	m_IOType :INT :=0;
	
	// counts after IO  is triggerd
	m_IOOnCounts :INT;
	
	// counts threshold indicating IO is trully triggerd
	m_IOOnCountThres :INT :=10;
END_VAR

METHOD check : BOOL
VAR_INPUT
	IOValue :BOOL;
END_VAR
check:=false;
IF (0=m_IOType and IOValue) OR (1=m_IOType AND NOT(IOValue)) THEN
	m_IOOnCounts := MIN(m_IOOnCounts +1, m_IOOnCountThres);
ELSE
	IF m_IOOnCounts>=m_IOOnCountThres THEN
		check:=TRUE;
	END_IF
	 m_IOOnCounts :=0;
END_IF
END_METHOD

METHOD init : BOOL
VAR_INPUT
	i_IOType :INT;
	i_triggerCounts:INT;
END_VAR
m_IOType:=i_IOType;
m_IOOnCountThres := i_triggerCounts;
END_METHOD

END_FUNCTION_BLOCK

// ---- FBs_Robots/FB_CartJoint.TcPOU
FUNCTION_BLOCK FB_CartJoint EXTENDS FB_JointBase
VAR_INPUT
END_VAR
VAR_OUTPUT
END_VAR
VAR
END_VAR

METHOD PUBLIC init : BOOL
VAR_INPUT
	i_jntIdx :INT;
	i_controlCycleTime :LREAL;
END_VAR
m_cycleTime := i_controlCycleTime;

// hardware parameters
m_motorEncoderRes :=GVL_CartJointParameters.g_incEncoderRes[i_jntIdx];
m_linkEncoderRes :=GVL_CartJointParameters.g_absEncoderRes[i_jntIdx];
m_motorReduction :=GVL_CartJointParameters.g_motorReduction[i_jntIdx];
m_linkEncoderReduction :=GVL_CartJointParameters.g_absEncoderReduction[i_jntIdx];
m_trqConst :=GVL_CartJointParameters.g_motorTrqConst[i_jntIdx];
m_maxCurrent :=GVL_CartJointParameters.g_motorMaxCurrent[i_jntIdx];
m_motorDir :=GVL_CartJointParameters.g_motorDir[i_jntIdx];								
m_linkEncoderDir :=GVL_CartJointParameters.g_asbEncoderDir[i_jntIdx];
m_minJntPos	:=GVL_CartJointParameters.g_minJntPos[i_jntIdx];
m_maxJntPos	:=GVL_CartJointParameters.g_maxJntPos[i_jntIdx];

//link encoder calibartion data
m_minLinkEncoder :=GVL_CartJointCaliData.g_minLinkEncoder[i_jntIdx] - m_linkEncoderDir*GVL_CartJointCaliData.g_linkEncLimitBuffer; // expand limit
m_maxLinkEncoder :=GVL_CartJointCaliData.g_maxLinkEncoder[ i_jntIdx] + m_linkEncoderDir*GVL_CartJointCaliData.g_linkEncLimitBuffer; // expand limit
m_caliLinkEncoder :=GVL_CartJointCaliData.g_caliLinkEncoder[i_jntIdx];
m_linkEncCaliJntPos :=GVL_CartJointCaliData.g_linkEncCaliJntPos[i_jntIdx];
m_linkEncZeroCross :=GVL_CartJointCaliData.g_linkEncZeroCross[i_jntIdx];
m_multiCycles :=GVL_CartJointCaliData.g_multipleCyclesJoint[i_jntIdx];

// convert cali link encoder if joint cross zero
IF 1=m_linkEncZeroCross THEN
	IF 1=m_linkEncoderDir AND m_caliLinkEncoder < m_minLinkEncoder THEN
		m_caliLinkEncoder := GVL_CartJointCaliData.g_caliLinkEncoder[i_jntIdx] + m_linkEncoderRes;
	ELSIF -1=m_linkEncoderDir AND m_caliLinkEncoder < m_maxLinkEncoder THEN
		m_caliLinkEncoder := GVL_CartJointCaliData.g_caliLinkEncoder[i_jntIdx] + m_linkEncoderRes;
	END_IF
END_IF

// macro data
m_trq2CurrentRatio:=m_motorDir * 1000.0/(m_trqConst*m_motorReduction);
m_current2TrqRatio:=m_motorDir * (m_trqConst*m_motorReduction)/1000.0;
m_linkEnc2PosRatio := 2*PI*m_linkEncoderDir/(m_linkEncoderReduction*m_linkEncoderRes);
m_motorEnc2PosRatio := 2*PI * m_motorDir/(m_motorReduction * m_motorEncoderRes);

// motor data init
m_curJntVel:=0;
m_curJntTrq :=0;
m_rawCurrent :=0;
m_filtCurrent :=0;
m_cmdJntVel :=0.0;
m_cmdJntTrq :=0.0;
m_cmdCurrent := 0.0;

// filter init
m_jntVelLpf.init(1, g_curJntVelLpfCutoffFreq, g_cartCtrlFreq);
m_linkVelLpf.init(1, g_curJntVelLpfCutoffFreq, g_cartCtrlFreq);
m_cmdTrqLpf.init(1, g_cmdJntTrqLpfCutoffFreq, g_cartCtrlFreq);
m_curTrqLpf.init(1, g_curJntTrqLpfCutoffFreq, g_cartCtrlFreq);

// driver init value
m_motorOutputs.m_controlWord:=DriverCtrlWord_INIT;
m_motorOutputs.m_opMode:=INT_TO_SINT(DriverOPMode_Pos);
m_motorOutputs.m_cmdCurrent:=0;
m_motorOutputs.m_cmdMotorEncoder:=m_motorInputs.m_motorEncoder;
END_METHOD

END_FUNCTION_BLOCK

// ---- FBs_StateControllers/FB_StateCtrlInit.TcPOU
// Brief: Master Arm Master Slave Control
FUNCTION_BLOCK PUBLIC FB_StateCtrlInit EXTENDS FB_MasterArmCtrlBase
VAR_INPUT
END_VAR
VAR_OUTPUT
END_VAR
VAR
	m_jnt7SelfCheckVel : LREAL :=180*g_deg2Rad;
	m_jnt7HalfMotionRange : LREAL := 1.75*PI+0.26;
	m_jnt7LimitErr :LREAL := 5*g_deg2Rad;
	m_jnt7CenterPos :LREAL;
	// 0: driver on; 1: joint 7 move to upper limit, 2: joint 7 mvoe to center
	m_initState :INT :=0;
END_VAR

// override this function in each exact controller
METHOD PROTECTED calcCmdJntPos : BOOL

VAR_IN_OUT CONSTANT
	i_slaveIdx :INT;
	i_shoulderPose :ST_Frame;
	i_masterArm :FB_MasterArm;
	i_slaveStatus :ST_SlaveStatus;
END_VAR

VAR
	centerVel:LREAL;
//	curJntPos:Vec7d;
END_VAR
IF m_isFinished THEN
	RETURN;
END_IF

CASE m_initState OF
	0:
		m_cmdJntPos := i_masterArm.curJntPos;
		IF i_masterArm.isEnabled(m_jntEnableFlag) = TRUE THEN
			m_initState :=1;
		END_IF
	1: 
		m_cmdJntPos[7] := m_cmdJntPos[7] + m_jnt7SelfCheckVel * g_armCtrlCycleTime;
		IF m_cmdJntPos[7]-i_masterArm.curJntPos[7] > m_jnt7LimitErr THEN
			m_cmdJntPos[7]:=i_masterArm.curJntPos[7];
			m_jnt7CenterPos :=m_cmdJntPos[7]-m_jnt7HalfMotionRange;
			m_initState :=2;
		END_IF
	2:
		centerVel :=LIMIT(-m_jnt7SelfCheckVel,(m_jnt7CenterPos-m_cmdJntPos[7])/g_armCtrlCycleTime,m_jnt7SelfCheckVel);
		m_cmdJntPos[7] := m_cmdJntPos[7] + centerVel * g_armCtrlCycleTime;
		IF ABS(m_jnt7CenterPos-i_masterArm.curJntPos[7]) < g_jntCtrlAngTolLow THEN
			m_isFinished :=TRUE;
		END_IF
END_CASE
END_METHOD

METHOD PUBLIC init : BOOL
VAR_IN_OUT CONSTANT
	i_masterArm	:FB_MasterArm;
END_VAR
VAR_IN_OUT 
	r_masterArmCtrlCmd :ST_ArmCtrlCmds;
END_VAR

VAR
	i:INT;
END_VAR
SUPER^.Init(i_masterArm,r_masterArmCtrlCmd);
m_initState :=0;
END_METHOD

END_FUNCTION_BLOCK

// ---- FBs_StateControllers/FB_StateCtrlHome.TcPOU
// Brief: Master Arm Home Posture
FUNCTION_BLOCK PUBLIC FB_StateCtrlHome EXTENDS FB_MasterArmCtrlBase
VAR_INPUT
END_VAR
VAR_OUTPUT
END_VAR
VAR
	m_homePlanner : FB_TrajMoveJ;
	
END_VAR

// override this function in each exact controller
METHOD PROTECTED calcCmdJntPos : BOOL
VAR_IN_OUT CONSTANT
	i_slaveIdx :INT;
	i_shoulderPose :ST_Frame;
	i_masterArm :FB_MasterArm;
	i_slaveStatus :ST_SlaveStatus;
END_VAR
VAR 
	i :INT;
	curJntVel :Vec7d;
END_VAR
// check if planner is ready
IF m_homePlanner.isGene = FALSE THEN
	calcCmdJntPos:=FALSE;
	RETURN;
END_IF

// traj plan
calcCmdJntPos :=m_homePlanner.evaluate(m_timePeriod, jntPos=> m_cmdJntPos, jntVel=>m_cmdJntVel, jntAcc=> m_cmdJntAcc);

// check if to terminate
curJntVel :=i_masterArm.curJntVel;
m_isFinished :=m_timePeriod > m_homePlanner.duration  AND norm(curJntVel)<7*g_jntStaticVelThres;
END_METHOD

METHOD PUBLIC init : BOOL
VAR_IN_OUT CONSTANT
	i_masterArm	:FB_MasterArm;
END_VAR
VAR_IN_OUT 
	r_masterArmCtrlCmd :ST_ArmCtrlCmds;
END_VAR

VAR
	i,j :INT;
	startJntPos,endJntPos :Vec7d;
END_VAR
SUPER^.Init(i_masterArm,r_masterArmCtrlCmd);

// traj plan
startJntPos:=i_masterArm.curJntPos;
FOR j:=1 TO 7 DO 
endJntPos[j]:=g_homePosture[i_masterArm.armIdx,j];
END_FOR
m_homePlanner.init(startJntPos,endJntPos,g_homeMaxjntVel,g_homeMaxjntAcc,g_homeMaxjntJerk);

// update commands to arm
copyCmds(r_masterArmCtrlCmd);
END_METHOD

END_FUNCTION_BLOCK

// ---- FBs_TrajectoryPlanning/FB_TrajMoveJ.TcPOU
FUNCTION_BLOCK FB_TrajMoveJ EXTENDS FB_TrajBase
VAR_OUTPUT
END_VAR
VAR
	// move vector in joint space
	m_startPos:Vec7d;
	m_targetPos:Vec7d;
	m_moveDir : Vec7d;
	m_moveDistance :LREAL;
	
	// doubleS planning for move distance
	m_doubleS :FB_BasicDoubleS;

END_VAR

METHOD evaluate : BOOL
VAR_INPUT
	t :LREAL;
END_VAR

VAR_OUTPUT
	jntPos,jntVel, jntAcc :vec7d;
END_VAR
VAR
	q,q_dot,q_ddot :LREAL;
	moveRange :Vec7d;
END_VAR
evaluate:=m_doubleS.evaluate(t,q=>q,q_dot=>q_dot, q_ddot=>q_dot);

IF evaluate =FALSE THEN
	RETURN;
END_IF

vecMultiNum(m_moveDir,q, moveRange);
vecAdd(moveRange, m_startPos,jntPos);
vecMultiNum(m_moveDir,q_dot, jntVel);
vecMultiNum( m_moveDir,q_ddot, jntAcc);
END_METHOD

METHOD init : BOOL
VAR_INPUT
	i_startJntPos :Vec7d;
	i_targetJntPos :Vec7d;
	i_maxJntVel : Vec7d;
	i_maxJntAcc : Vec7d;
	i_maxJntJerk :Vec7d;
END_VAR
VAR 
	i:INT;
	maxV, maxA, maxJ :LREAL;
	q:ARRAY[1..2] OF LREAL;
	v:ARRAY[1..2] OF LREAL;
END_VAR
m_startPos:=i_startJntPos;
m_targetPos:=i_targetJntPos;
vecSub(i_targetJntPos, i_startJntPos, m_moveDir);
m_moveDistance := norm(m_moveDir);

IF(m_moveDistance<g_smallNum) THEN
	vecMultiNum(g_onesVec7d,1/7, m_moveDir);;
ELSE
	vecMultiNum( m_moveDir,1/m_moveDistance, m_moveDir);
END_IF

// determian max vel/acc/jerk
maxV:=g_largeNum;
maxA:=g_largeNum;
maxJ:=g_largeNum;
FOR i :=1 TO 7 DO 
	IF ABS(m_moveDir[i])>g_smallNum THEN
		maxV := MIN (maxV, ABS(i_maxJntVel[i]/m_moveDir[i]));
		maxA := MIN (maxA, ABS(i_maxJntAcc[i]/m_moveDir[i]));
		maxJ := MIN (maxJ, ABS(i_maxJntJerk[i]/m_moveDir[i]));
	END_IF
END_FOR

// planning for moving distance
q[1]:=0;
q[2]:=m_moveDistance;
v[1]:=0;
v[2]:=0;
m_doubleS.init(q,v, maxV, maxA, maxJ);
m_duration:=m_doubleS.duration;
m_isGenerated:=m_doubleS.isGene;
END_METHOD

END_FUNCTION_BLOCK

// ---- FBs_TrajectoryPlanning/FB_trajBase.TcPOU
FUNCTION_BLOCK FB_trajBase
VAR_INPUT
END_VAR
VAR_OUTPUT
END_VAR
VAR
	// total trajectory duration
	m_duration :LREAL:=0;
	
	// flag is trajectory is init successfully 
	m_isGenerated : BOOL :=FALSE;
END_VAR

PROPERTY duration : lreal
GET
duration:=m_duration;
END_GET
END_PROPERTY

PROPERTY isGene : bool
GET
isGene:=m_isGenerated;
END_GET
END_PROPERTY

END_FUNCTION_BLOCK

// ---- FBs_TrajectoryPlanning/FB_BasicDoubleS.TcPOU
// reference: Trajectory planning for automation machines and robots
FUNCTION_BLOCK FB_BasicDoubleS EXTENDS FB_trajBase
VAR_INPUT
END_VAR
VAR_OUTPUT
END_VAR
VAR
	// endpoints position AND velocity
	m_q :ARRAY[1..2] OF LREAL;
	m_v :ARRAY[1..2] OF LREAL;
	
	// traj constraint
	m_maxV :LREAL:=0;
	m_maxA :LREAL:=0;
	m_maxJ :LREAL:=0;
	
	// acceleration duration
	m_Taj :LREAL :=0;
	m_Ta :LREAL :=0;
	
	// constant velocity duration
	m_Tv :LREAL :=0;
	
	// deceleration duration
	m_Tdj :LREAL :=0;
	m_Td:LREAL :=0;
	
	// traj sign
	m_sign : LREAL :=1;
	
	// trajectory parmaters
	m_limitAcc :LREAL :=0;
	m_limitDec :LREAL :=0;
	m_limitVel :LREAL :=0;
END_VAR

METHOD PUBLIC evaluate : BOOL
VAR_INPUT
	t :LREAL;
END_VAR

VAR_OUTPUT
	q,q_dot,q_ddot :LREAL;
END_VAR
VAR
	q0,q1,v0,v1:LREAL;
END_VAR
IF FALSE = m_isGenerated THEN
	evaluate := FALSE;
	RETURN;
END_IF

q:=0;
q_dot:=0;
q_ddot:=0;
q0:=m_q[1];
q1:=m_q[2];
v0:=m_v[1];
v1:=m_v[2];

IF t<=0 THEN
	q:=q0;
	q_dot:=v0;
	q_ddot:=0;
ELSIF m_Taj>0 AND  t<=m_Taj THEN
	q:=q0+v0*t+m_maxJ*EXPT(t,3)/6;
	q_dot:=v0+m_maxJ*EXPT(t,2)/2;
	q_ddot:=m_maxJ*t;
ELSIF m_Ta>2*m_Taj AND  t<=m_Ta-m_Taj THEN
	q:=q0+v0*t+m_limitAcc*(3*EXPT(t,2)-3*m_Taj*t+EXPT(m_Taj,2))/6;
	q_dot:=v0+m_limitAcc*(t-m_Taj/2);
	q_ddot:=m_limitAcc;
ELSIF m_Taj>0 AND  t<=m_Ta THEN
	q:=q0+(v0+m_limitVel)*m_Ta/2-m_limitVel*(m_Ta-t)+m_maxJ*EXPT(m_Ta-t,3)/6;
	q_dot:=m_limitVel-m_maxJ*EXPT(m_Ta-t,2)/2;
	q_ddot:=m_maxJ*(m_Ta-t);
ELSIF m_Tv>0 AND  t<=m_Ta+m_Tv THEN
	q:=q0+(v0+m_limitVel)*m_Ta/2+m_limitVel*(t-m_Ta);
	q_dot:=m_limitVel;
	q_ddot:=0;
ELSIF m_Tdj>0 AND  t<=m_Ta+m_Tv+m_Tdj THEN
	q:=q1-(m_limitVel+v1)*m_Td/2+m_limitVel*(t-m_duration+m_Td)-m_maxJ*EXPT(t-m_duration+m_Td,3)/6;
	q_dot:=m_limitVel-m_maxJ*EXPT(t-m_duration+m_Td,2)/2;
	q_ddot:=-m_maxJ*(t-m_duration+m_Td);
ELSIF m_Td>2*m_Tdj AND  t<=m_duration-m_Tdj THEN
	q:=q1-(m_limitVel+v1)*m_Td/2+m_limitVel*(t-m_duration+m_Td)+m_limitDec*(3*expt(t-m_duration+m_Td,2)-3*m_Tdj*(t-m_duration+m_Td)+m_Tdj*m_Tdj)/6;
	q_dot:=m_limitVel+m_limitDec*(t-m_duration+m_Td-m_Tdj/2);
	q_ddot:=m_limitDec;
ELSIF m_Tdj>0 AND  t<=m_duration THEN
	q:=q1-v1*(m_duration-t)-m_maxJ*EXPT(m_duration-t,3)/6;
	q_dot:=v1+m_maxJ*EXPT(m_duration-t,2)/2;
	q_ddot:=-m_maxJ*(m_duration-t);
ELSIF t>m_duration THEN
	q:=q1;
	q_dot:=v1;
	q_ddot:=0;
END_IF

q:=m_sign*q;
q_dot:=m_sign*q_dot;
q_ddot:=m_sign*q_dot;
evaluate := TRUE;
END_METHOD

METHOD PUBLIC init : BOOL
VAR_INPUT
	q :ARRAY[1..2] OF LREAL;
	v :ARRAY[1..2] OF LREAL;
	maxV :LREAL;
	maxA :LREAL;
	maxJ :LREAL;
END_VAR
VAR
	q0,q1,v0,v1,h,Delta :LREAL;
	recursiveStep :LREAL :=0.7;
	maxRecursiveTime :INT :=20;
	recursiveTime :INT :=0;
END_VAR
//normalize computation AND parameters
m_isGenerated:=FALSE;
IF q[2]=q[1] THEN
	m_sign:=1;
else
	m_sign:=(q[2]-q[1])/ABS(q[2]-q[1]);
END_IF
m_q[1]:=m_sign*q[1];
m_q[2]:=m_sign*q[2];
m_v[1]:=m_sign*v[1];
m_v[2]:=m_sign*v[2];
m_maxV:=maxV;
m_maxA:=maxA;
m_maxJ:=maxJ;

// set initial and final parameters
q0:=m_q[1];
q1:=m_q[2];
v0:=m_v[1];
v1:=m_v[2];
h:=q1-q0;

// check if traj is feasible
IF trajCheck(q1-q0,v0,v1,maxA,maxJ)=FALSE THEN 
	init :=FALSE;
	RETURN;
END_IF

// if initial and final position is same
IF ABS(q1-q0)<g_smallNum THEN
	m_Tv:=g_smallNum;
	m_duration:=g_smallNum;
	m_isGenerated:=TRUE;
	return;
END_IF

// assuming tha maxV are reached and compute the time intervel of constant velocity
// maxA not reached
IF maxA*maxA>(maxV-v0)*maxJ THEN
	m_Taj:=SQRT((maxV-v0)/maxJ);
	m_Ta:=2*m_Taj;
	m_limitAcc:=m_Taj*maxJ;
// maxA reached
else
	m_Taj:=maxA/maxJ;
	m_Ta:=m_Taj+(maxV-v0)/maxA;
	m_limitAcc:=maxA;
END_IF

// minA not reached
IF maxA*maxA>(maxV-v1)*maxJ THEN
	m_Tdj:=SQRT((maxV-v1)/maxJ);
	m_Td:=2*m_Tdj;
	m_limitDec:=-m_Tdj*maxJ;
// minA reached
else
	m_Tdj:=maxA/maxJ;
	m_Td:=m_Tdj+(maxV-v1)/maxA;
	m_limitDec:=-maxA;
END_IF
m_Tv:=(q1-q0)/maxV-m_Ta*(1+v0/maxV)/2-m_Td*(1+v1/maxV)/2;

// maxV reached
IF m_Tv>0 THEN
	m_limitVel:=maxV;
	m_isGenerated:=TRUE;
// maxV not reached, in this case, maxA must reach
else
	m_Tv:=0;
	recursiveTime:=0;
	WHILE(m_isGenerated=FALSE AND recursiveTime<maxRecursiveTime) DO
		m_Taj:=maxA/maxJ;
		m_Tdj:=maxA/maxJ;
		Delta:=EXPT(maxA,4)/EXPT(maxJ,2)+2*(v0*v0+v0*v1)+maxA*(4*h-2*maxA*(v0+v1)/maxJ);
		m_Ta:=(maxA*maxA/maxJ-2*v0+SQRT(Delta))/(2*maxA);
		m_Td:=(maxA*maxA/maxJ-2*v1+SQRT(Delta))/(2*maxA);
		IF(m_Ta<0 AND v0>v1) THEN
			m_Taj:=0;
			m_Ta:=0;
			m_Td:=2*h/(v1+v0);
			m_Tdj:=(maxJ*h-SQRT(maxJ*(maxJ*h*h+EXPT(v0+v1,2)*(v1-v0))))/(maxJ*(v1+v0));
			m_isGenerated:=TRUE;
		ELSIF(m_Td<0 AND v1>v0) THEN
			m_Tdj:=0;
			m_Td:=0;
			m_Ta:=2*h/(v1+v0);
			m_Taj:=(maxJ*h-SQRT(maxJ*(maxJ*h*h-EXPT(v0+v1,2)*(v1-v0))))/(maxJ*(v1+v0));
			m_isGenerated:=TRUE;
		END_IF

		IF m_Ta>=2*m_Taj AND m_Td>=2*m_Tdj THEN
			m_isGenerated:=TRUE;
		END_IF

		IF m_isGenerated=TRUE THEN
			m_limitAcc:=maxJ*m_Taj;
			m_limitDec:=-maxJ*m_Tdj;
			m_limitVel:=v0+(m_Ta-m_Taj)*m_limitAcc;
			EXIT;       
		END_IF
		recursiveTime:=recursiveTime+1;
		maxA:=maxA*recursiveStep;
	END_WHILE
END_IF

// total duration
m_duration:=m_Ta+m_Tv+m_Td;
END_METHOD

// check if the trajectory is feasible
METHOD PROTECTED trajCheck : BOOL
VAR_INPUT
	h : LREAL;
	v0 : LREAL;
	v1 : LREAL;
	maxA : LREAL;
	maxJ : LREAL;
END_VAR
VAR
	T1,T2,dis,t :LREAL;
END_VAR
T1:=SQRT(ABS(v1-v0)/maxJ);
T2:=maxA/maxJ;
t:=MIN(T1,T2);
IF t<T2 THEN
	dis:=t*ABS(v0+v1);
else
	dis:=ABS(v0+v1)*(t+ABS(v1-v0)/maxA)/2;
END_IF

IF ABS(h)>=dis THEN 
	trajCheck:=TRUE;
else
	trajCheck:=FALSE;
END_IF
END_METHOD

END_FUNCTION_BLOCK

// ---- AgiMaths/MatrixLib/vecAdd.TcPOU
// C = A + B;
FUNCTION vecAdd : BOOL
VAR_IN_OUT CONSTANT
	vecA :ARRAY[*] OF LREAL;
	vecB :ARRAY[*] OF LREAL;
END_VAR

VAR_IN_OUT 
	vecC :ARRAY[*] OF LREAL;
END_VAR

VAR
	m :DINT;
	i:DINT;
 
END_VAR

m:=UPPER_BOUND(VecA,1);
ASSERT(UPPER_BOUND(VecB,1)=m);
ASSERT(UPPER_BOUND(VecC,1)=m);

FOR i:=1 TO m DO
	vecC[i]:=vecA[i]+vecB[i];
END_FOR

END_FUNCTION

// ---- FBs_StateControllers/FB_StateCtrlStandBy.TcPOU
// Brief: Master Arm Standby
FUNCTION_BLOCK PUBLIC FB_StateCtrlStandBy EXTENDS FB_MasterArmCtrlBase
VAR_INPUT
END_VAR
VAR_OUTPUT
END_VAR
VAR
END_VAR

METHOD PUBLIC init : BOOL
VAR_IN_OUT CONSTANT
	i_masterArm	:FB_MasterArm;
END_VAR
VAR_IN_OUT 
	r_masterArmCtrlCmd :ST_ArmCtrlCmds;
END_VAR
// check if to hold the command joint position unchanged
m_holdLastCmds := checkToHoldLastCmds(i_masterArm);

// init
SUPER^.Init(i_masterArm,r_masterArmCtrlCmd);

m_jntOPMode[4] := DriverOPMode_PosTrq;
m_jntOPMode[5] := DriverOPMode_PosTrq;
m_jntOPMode[6] := DriverOPMode_PosTrq;
m_jntOPMode[7] := DriverOPMode_PosTrq;
END_METHOD

END_FUNCTION_BLOCK

// ---- FBs_StateControllers/FB_StateCtrlMatching.TcPOU
// Brief: Master Arm Orientation Matching
FUNCTION_BLOCK PUBLIC FB_StateCtrlMatching EXTENDS FB_MasterArmCtrlBase
VAR_INPUT
END_VAR
VAR_OUTPUT
END_VAR
VAR
	// master-slave orientation match threshold
	m_matchAngleThres :LREAL := 2*g_deg2Rad;
	
	m_cmdRotInMonitor :Mat3d;
	
	m_initSolvedJntPos, m_iteSovlvedJntPos :Vec7d;
	m_IKSuccess :BOOL;
	
	m_matchTrajPlanner : FB_TrajMoveJ;
	m_targetJntPos :Vec7d;
	
	m_maxMatchJntVel:Vec7d:=[1.0, 1.0, 1.0, 2*pi, 3*pi, 3*pi, 5*pi];
	m_maxMatchJntAcc:Vec7d:=[1.0, 1.0, 1.0,  8*pi, 12*pi, 12*pi, 20*pi];
	m_maxMatchJntJerk:Vec7d:=[7(100.0)];
	
	m_rotErrAng :LREAL;

END_VAR

// override this function in each exact controller
METHOD PROTECTED calcCmdJntPos : BOOL

VAR_IN_OUT CONSTANT
	i_slaveIdx :INT;
	i_shoulderPose :ST_Frame;
	i_masterArm :FB_MasterArm;
	i_slaveStatus :ST_SlaveStatus;
END_VAR
var 
	i,j : INT;

	mq4,mq5,mq6,mq7:LREAL;
	q4,q5,q6,q7:LREAL;

	rotErr:Mat3d;
	wristRotInJnt3, wristRotInJnt4 :Mat3d;
	rot, invRot :Mat3d;
	cycleNum:INT;
	
	jnt4MoveRange:LREAL;
	jnt5Bias, jnt4MoveScale :LREAL;
	
	cmdJntErr:Vec7d;

END_VAR
IF m_IKSuccess THEN 
	// check if planner is ready
	IF  m_matchTrajPlanner.isGene = FALSE THEN
		RETURN;
	END_IF
	
	// traj plan
	calcCmdJntPos :=m_matchTrajPlanner.evaluate(m_timePeriod, jntPos=> m_cmdJntPos, jntVel=>m_cmdJntVel, jntAcc=> m_cmdJntAcc);
	
	vecSub(m_targetJntPos, m_cmdJntPos, cmdJntErr);
	
	matTranspose(i_masterArm.curCartPose.m_rot, invRot);
	matMultiply(invRot, m_cmdCartPose.m_rot, rotErr);
	rot2AngAxis(rotErr, angle=>m_rotErrAng,axis=>);
	m_isFinished := m_timePeriod > m_matchTrajPlanner.duration AND  norm(cmdJntErr)<g_jntCtrlAngTolHigh;
	
	RETURN;
END_IF

// command rotation in monitor
m_cmdRotInMonitor := i_slaveStatus.m_curArmPose[i_slaveIdx].m_rot;

// command rotation in master arm base
matTranspose(i_shoulderPose.m_rot, invRot);
matMultiply(invRot, m_cmdRotInMonitor, m_cmdCartPose.m_rot);
m_cmdCartPose.m_pos:= i_masterArm.curCartPose.m_pos;

// calculate current orientation error
matTranspose(i_masterArm.curCartPose.m_rot, invRot);
matMultiply(invRot, m_cmdCartPose.m_rot, rotErr);
rot2AngAxis(rotErr, angle=>m_rotErrAng,axis=>);

// try IK with optimized posture
rot:=calcJnt3Rotation(m_cmdJntPos[1],m_cmdJntPos[2],m_cmdJntPos[3]);
matTranspose(rot, invRot);
matMultiply(invRot, m_cmdCartPose.m_rot, wristRotInJnt3);
IF 1=i_masterArm.armIdx THEN
	m_IKSuccess := leftWristOptIK(wristRotInJnt3,q4=>q4, q5=>q5, q6=>q6, q7=>q7);
ELSE
	m_IKSuccess := rightWristOptIK(wristRotInJnt3,q4=>q4, q5=>q5, q6=>q6, q7=>q7);
END_IF

// try IK with joint4 at minimal limit
IF NOT m_IKSuccess THEN
	q4:= GVL_ArmJointParameters.g_minJntPos[i_masterArm.armIdx,4];
	
	rot:=calcJnt4Rotation(m_cmdJntPos[1],m_cmdJntPos[2],m_cmdJntPos[3],q4);
	matTranspose(rot, invRot);
	matMultiply(invRot, m_cmdCartPose.m_rot, wristRotInJnt4);
	m_IKSuccess := wristIK(wristRotInJnt4,i_masterArm, q5=>q5, q6=>q6, q7=>q7);
END_IF

// try IK with joint4 at maximum limit
IF NOT m_IKSuccess THEN
	q4:= GVL_ArmJointParameters.g_maxJntPos[i_masterArm.armIdx,4];
	
	rot:=calcJnt4Rotation(m_cmdJntPos[1],m_cmdJntPos[2],m_cmdJntPos[3],q4);
	matTranspose(rot, invRot);
	matMultiply(invRot, m_cmdCartPose.m_rot, wristRotInJnt4);
	m_IKSuccess := wristIK(wristRotInJnt4,i_masterArm, q5=>q5, q6=>q6, q7=>q7);
END_IF

// minimize joint4 move angle
IF m_IKSuccess THEN
	
	// minimize based on join5 posture
	jnt4MoveRange :=  i_masterArm.jnt4LinkToMotor(m_targetJntPos[2],m_targetJntPos[3],q4)-i_masterArm.curJntPos[4];
	jnt5Bias :=  LIMIT (0, ABS(q5-pi), pi/2);
	jnt4MoveRange := jnt4MoveRange * ABS(COS(jnt5Bias));
	
	// minimize based on cartesian error
	IF ABS(m_rotErrAng)< 5.0 * g_deg2Rad THEN
		jnt4MoveRange := 0.0;
	END_IF
	
	mq4:=  i_masterArm.jnt4MotorToLink(m_targetJntPos[2],m_targetJntPos[3],i_masterArm.curJntPos[4] + jnt4MoveRange) ;
	
	rot:=calcJnt4Rotation(m_cmdJntPos[1],m_cmdJntPos[2],m_cmdJntPos[3],mq4);
	matTranspose(rot, invRot);
	matMultiply(invRot, m_cmdCartPose.m_rot, wristRotInJnt4);
	IF wristIK(wristRotInJnt4,i_masterArm, q5=>mq5, q6=>mq6, q7=>mq7) THEN
		q4:=mq4;
		q5:=mq5;
		q6:=mq6;
		q7:=mq7;
	END_IF
END_IF

// traj plan
IF m_IKSuccess THEN 
	m_targetJntPos:=m_cmdJntPos;
	m_targetJntPos[4]:=i_masterArm.jnt4LinkToMotor(m_targetJntPos[2],m_targetJntPos[3],q4);
	m_targetJntPos[5]:=q5;
	m_targetJntPos[6]:=q6;
	
	// roll flip handle
	i_masterArm.flipGripper(rollFlipHandle(i_masterArm.armIdx,i_masterArm.curJntPos[7], q7, o_cmdJntPos7 =>m_targetJntPos[7]));
	
	// no match for rotate joint if instrument is ultrasonic knife
	IF MasterArmControl.m_masterRobot.m_USKnifeRotClutch[i_slaveIdx] THEN
		m_targetJntPos[7] := i_masterArm.curJntPos[7];
	END_IF

	m_matchTrajPlanner.init(m_cmdJntPos,m_targetJntPos,m_maxMatchJntVel,m_maxMatchJntAcc,m_maxMatchJntJerk);
	m_timePeriod :=0;
END_IF
END_METHOD

// calculate joint3 rotation in arm coordinate
(*armDH=[   0      0   q1      d1;
            -deg90  0   q2      0;
            0       a3  q3      0];*)
METHOD PROTECTED calcJnt3Rotation : Mat3d
VAR_INPUT CONSTANT
	q1:LREAL;
	q2:LREAL;
	q3:LREAL;
END_VAR

VAR
	c1,c2,c3,s1,s2,s3,c23,s23 :LREAL;
END_VAR
// !Convert active joint position to DH model for kinematic calculation
q3:=q3-q2;  //q3=q8-q2

c1:=COS(q1);
c2:=COS(q2);
c3:=COS(q3);

s1:=SIN(q1);
s2:=SIN(q2);
s3:=SIN(q3);

c23:=COS(q2+q3);
s23:=SIN(q2+q3);

calcJnt3Rotation[1,1]:= c23*c1;
calcJnt3Rotation[2,1]:= c23*s1;
calcJnt3Rotation[3,1]:= -s23;

calcJnt3Rotation[1,2]:= -s23*c1;
calcJnt3Rotation[2,2]:= -s23*s1;
calcJnt3Rotation[3,2]:= -c23;

calcJnt3Rotation[1,3]:= -s1;
calcJnt3Rotation[2,3]:= c1;
calcJnt3Rotation[3,3]:=0;
END_METHOD

// calculate joint3 rotation in arm coordinate
(*[   0      0   q1      d1;
	-deg90  0   q2      0;
	0       a3  q3      0;
	 -deg90  a4  q4      d4]
*)
METHOD PROTECTED calcJnt4Rotation : Mat3d
VAR_INPUT
	q1 :LREAL;
	q2 :LREAL;
	q3 :LREAL;
	q4 :LREAL;// already at the link side
END_VAR

VAR
	c1,c2,c3,c4, s1,s2,s3,s4,c23,s23 :LREAL;
END_VAR
// !Convert active joint position to DH model for kinematic calculation
//q4:=q4+q3-q2-pi/2;//q4DH=q4motor+q8-q2-90;  
q3:=q3-q2;  //q3=q8-q2

c1:=COS(q1);
c2:=COS(q2);
c3:=COS(q3);
c4:=COS(q4);

s1:=SIN(q1);
s2:=SIN(q2);
s3:=SIN(q3);
s4:=SIN(q4);

c23:=COS(q2+q3);
s23:=SIN(q2+q3);

calcJnt4Rotation[1,1]:= s1*s4 + c4*c1*c23;
calcJnt4Rotation[2,1]:= - c1*s4 + c4*s1*c23;
calcJnt4Rotation[3,1]:= -s23*c4;

calcJnt4Rotation[1,2]:= c4*s1 - s4*c1*c23;
calcJnt4Rotation[2,2]:= -s4*s1*c23 - c1*c4;
calcJnt4Rotation[3,2]:=   s23*s4;

calcJnt4Rotation[1,3]:= -s23*c1;
calcJnt4Rotation[2,3]:= -s23*s1;
calcJnt4Rotation[3,3]:=-c23;
END_METHOD

PROPERTY IKSuccess : BOOL
GET
IKSuccess := m_IKSuccess;
END_GET
END_PROPERTY

METHOD PUBLIC init : BOOL
VAR_IN_OUT CONSTANT
	i_masterArm	:FB_MasterArm;
END_VAR
VAR_IN_OUT 
	r_masterArmCtrlCmd :ST_ArmCtrlCmds;
END_VAR
// check if to hold the command joint position unchanged
m_holdLastCmds := checkToHoldLastCmds(i_masterArm);

// init
SUPER^.Init(i_masterArm,r_masterArmCtrlCmd);

m_jntOPMode[4]:=DriverOPMode_PosTrq;
m_jntOPMode[5]:=DriverOPMode_PosTrq;
m_jntOPMode[6]:=DriverOPMode_PosTrq;
m_jntOPMode[7]:=DriverOPMode_PosTrq;

m_IKSuccess:=FALSE;
m_targetJntPos:=m_cmdJntPos;

// update commands to arm
copyCmds(r_masterArmCtrlCmd);
END_METHOD

// calculate command wrist joint position with an optimized posture
(*wristDH=[   -deg90  a4  q4      d4;
            deg90   0   q5      0;
            -deg90  0   q6      0;
            deg90   0   q7      0];*)
// set q6 = -pi/2 for desired posture
(* wristRot = 
[ COS(q7)*SIN(q4) - COS(q4)*SIN(q5)*SIN(q7), - SIN(q4)*SIN(q7) - COS(q4)*COS(q7)*SIN(q5), -COS(q4)*COS(q5)]
[                           cos(q5)*sin(q7),                             cos(q5)*cos(q7),         -sin(q5)]
[ cos(q4)*cos(q7) + sin(q4)*sin(q5)*sin(q7),   cos(q7)*sin(q4)*sin(q5) - cos(q4)*sin(q7),  cos(q5)*sin(q4)]
*)
METHOD PROTECTED leftWristOptIK : BOOL
VAR_IN_OUT CONSTANT
	i_cmdRot :Mat3d;
END_VAR
VAR_OUTPUT
	q4 :LREAL;
	q5 :LREAL;
	q6 :LREAL;
	q7 :LREAL;
END_VAR

VAR
	q51,q52 :LREAL;
	s4,c4,s5,c5,s7,c7:LREAL;
	q4UnreachPosMin: LREAL :=-pi/2;
	q4UnreachPosMax: LREAL :=45*g_deg2Rad;
	
END_VAR
q6:=-PI/2;
// q5 = [pi-135deg, pi+135deg]
q5 := ASIN(-i_cmdRot[2,3]);
q5:= PI-q5;

// q5=3pi/2 or q5=pi/2
IF ABS(q5-3*PI/2)<g_smallAng OR ABS(q5-PI/2)<g_smallAng THEN
	q4:= -pi;
	s7:= -i_cmdRot[1,1]/(COS(q4)*SIN(q5));
	c7:= i_cmdRot[3,1]/COS(q4);
	q7:=atan2(s7,c7);
	leftWristOptIK:=TRUE;
	RETURN;
END_IF

// solution one 
c5 :=COS(q5);
s7:=i_cmdRot[2,1]/c5;
c7:= i_cmdRot[2,2]/c5;
q7:=atan2(s7,c7);

//q4=[-pi/2-225deg, -pi/2]
c4 := -i_cmdRot[1,3]/c5;
s4:= i_cmdRot[3,3]/c5;
q4:=atan2(s4,c4);
IF q4> GVL_ArmJointParameters.g_minJntPos[1,4] AND q4<GVL_ArmJointParameters.g_maxJntPos[1,4] THEN
	leftWristOptIK:=TRUE;
	RETURN;
ELSIF q4> GVL_ArmJointParameters.g_maxJntPos[1,4] AND q4-2*pi> GVL_ArmJointParameters.g_minJntPos[1,4] THEN
	q4:=q4-2*PI;
	leftWristOptIK:=TRUE;
	RETURN;
END_IF

// solution2
IF q5 > pi THEN
	q5 := 3*PI-q5;
ELSE
	q5:= pi-q5;
END_IF
IF q5 > GVL_ArmJointParameters.g_maxJntPos[1,5] OR q5<GVL_ArmJointParameters.g_minJntPos[1,5] THEN
	leftWristOptIK:=FALSE;
	RETURN;
END_IF

c5 :=COS(q5);
s7:=i_cmdRot[2,1]/c5;
c7:= i_cmdRot[2,2]/c5;
q7:=atan2(s7,c7);

c4 := -i_cmdRot[1,3]/c5;
s4:= i_cmdRot[3,3]/c5;
q4:=atan2(s4,c4);
IF q4> GVL_ArmJointParameters.g_minJntPos[1,4] AND q4<GVL_ArmJointParameters.g_maxJntPos[1,4] THEN
	leftWristOptIK:=TRUE;
	RETURN;
ELSIF q4> GVL_ArmJointParameters.g_maxJntPos[1,4] AND q4-2*pi< GVL_ArmJointParameters.g_minJntPos[1,4] THEN
	q4:=q4-2*PI;
	leftWristOptIK:=TRUE;
	RETURN;
END_IF
END_METHOD

// calculate command wrist joint position with an optimized posture
(*wristDH=[   -deg90  a4  q4      d4;
            deg90   0   q5      0;
            -deg90  0   q6      0;
            deg90   0   q7      0];*)
// set q6 = pi/2 for desired posture
(* wristRot = 
[ - cos(q7)*sin(q4) - cos(q4)*sin(q5)*sin(q7), sin(q4)*sin(q7) - cos(q4)*cos(q7)*sin(q5),  cos(q4)*cos(q5)]
[                             cos(q5)*sin(q7),                           cos(q5)*cos(q7),          sin(q5)]
[   sin(q4)*sin(q5)*sin(q7) - cos(q4)*cos(q7), cos(q4)*sin(q7) + cos(q7)*sin(q4)*sin(q5), -cos(q5)*sin(q4)]
 
*)
METHOD PROTECTED rightWristOptIK : BOOL
VAR_IN_OUT CONSTANT
	i_cmdRot :Mat3d;
END_VAR
VAR_OUTPUT
	q4 :LREAL;
	q5 :LREAL;
	q6 :LREAL;
	q7 :LREAL;
END_VAR

VAR
	q51,q52 :LREAL;
	s4,c4,s5,c5,s7,c7:LREAL;
	q4UnreachPosMin: LREAL :=-pi/2;
	q4UnreachPosMax: LREAL :=45*g_deg2Rad;
	
END_VAR
q6:=PI/2;
// q5 = [pi-135deg, pi+135deg]
q5 := ASIN(i_cmdRot[2,3]);
q5:= PI-q5;

// q5=3pi/2 or q5=pi/2
IF ABS(q5-3*PI/2)<g_smallAng OR ABS(q5-PI/2)<g_smallAng THEN
	q4:= 0;
	s7:= -i_cmdRot[1,1]/(COS(q4)*SIN(q5));
	c7:= -i_cmdRot[3,1]/COS(q4);
	q7:=atan2(s7,c7);
	rightWristOptIK:=TRUE;
	RETURN;
END_IF

// solution one 
c5 :=COS(q5);
s7:=i_cmdRot[2,1]/c5;
c7:= i_cmdRot[2,2]/c5;
q7:=atan2(s7,c7);

//q4=[-pi/2, -pi/2+225deg]
c4 := i_cmdRot[1,3]/c5;
s4:= -i_cmdRot[3,3]/c5;
q4:=atan2(s4,c4);
IF q4> GVL_ArmJointParameters.g_minJntPos[2,4] AND q4<GVL_ArmJointParameters.g_maxJntPos[2,4] THEN
	rightWristOptIK:=TRUE;
	RETURN;
END_IF

// solution2
IF q5 > pi THEN
	q5 := 3*PI-q5;
ELSE
	q5:= pi-q5;
END_IF
IF q5 > GVL_ArmJointParameters.g_maxJntPos[1,5] OR q5<GVL_ArmJointParameters.g_minJntPos[1,5] THEN
	rightWristOptIK:=FALSE;
	RETURN;
END_IF

c5 :=COS(q5);
s7:=i_cmdRot[2,1]/c5;
c7:= i_cmdRot[2,2]/c5;
q7:=atan2(s7,c7);

//q4=[-pi/2, -pi/2+225deg]
c4 := i_cmdRot[1,3]/c5;
s4:= -i_cmdRot[3,3]/c5;
q4:=atan2(s4,c4);
IF q4> GVL_ArmJointParameters.g_minJntPos[2,4] AND q4<GVL_ArmJointParameters.g_maxJntPos[2,4] THEN
	rightWristOptIK:=TRUE;
	RETURN;
END_IF
END_METHOD

METHOD PROTECTED rollFlipHandle : BOOL
VAR_INPUT
	i_armIdx:INT;
	i_curJntPos7 :LREAL;
	i_initCmdJntPos7 :LREAL;
END_VAR
VAR_OUTPUT
	o_cmdJntPos7 :LREAL;
END_VAR

VAR
	solFeasible1,solFeasible2 :BOOL;
	solIdx :INT:=0;
	halfcycleNum1, halfcycleNum2:INT;
	solution1, solution2 :LREAL;
END_VAR
// this part is used to drive gripper back near center, in case that gripper roll is stuck near limit
// TODO: remove after gripper roll has infinite motion range
IF NOT (MasterArmControl.m_masterInputDataPool.m_cartStatus.m_surgonReady) THEN
	o_cmdJntPos7:=i_initCmdJntPos7;
	rollFlipHandle:=FALSE;
	RETURN;
END_IF

// handle multiple cycles of joint7
// find the first solution within pi from current position
halfcycleNum1 := LREAL_TO_INT((i_curJntPos7 - i_initCmdJntPos7)/pi);
solution1 := halfcycleNum1 * pi + i_initCmdJntPos7;

// solution2
IF solution1 > i_curJntPos7 THEN
	solution2 := solution1 - PI;
	halfcycleNum2 := halfcycleNum1 - 1;
ELSE
	solution2 := solution1 + PI;
	halfcycleNum2 := halfcycleNum1 + 1;
END_IF

//choose the solution which is closer to current q7 which can achive orientation match with a max pi/2 degree
// NOTE: There maybe risk this joint7 is stuck at limit, which can be solved after joint7 has infinite rotation angle,
solFeasible1:=solution1> GVL_ArmJointParameters.g_minJntPos[i_armIdx,7] AND solution1< GVL_ArmJointParameters.g_maxJntPos[i_armIdx,7];
solFeasible2:=solution2> GVL_ArmJointParameters.g_minJntPos[i_armIdx,7] AND solution2< GVL_ArmJointParameters.g_maxJntPos[i_armIdx,7];
IF solFeasible1 AND solFeasible2 THEN
	IF ABS(solution1-i_curJntPos7) < ABS(solution2-i_curJntPos7)  THEN
		solIdx:=1;
	ELSE
		solIdx:=2;
	END_IF
ELSIF solFeasible1 AND NOT(solFeasible2) THEN
	solIdx:=1;
ELSIF solFeasible2 AND NOT(solFeasible1) THEN
	solIdx:=2;
ELSE
	solIdx:=0;
END_IF

IF solIdx = 1 THEN
	o_cmdJntPos7 := solution1;
	rollFlipHandle:= ((ABS(halfcycleNum1) MOD 2) = 1);
ELSIF solIdx =2 THEN
	o_cmdJntPos7 := solution2;
	rollFlipHandle:= ((ABS(halfcycleNum2) MOD 2) = 1);
ELSE
	o_cmdJntPos7:=i_initCmdJntPos7;
	rollFlipHandle:=FALSE;
END_IF
END_METHOD

// calculate position of joint 5/6/7 
(*wristDH=[   deg90   0   q5      0;
            -deg90  0   q6      0;
            deg90   0   q7      0];*)
(* wristRot = 
[ cos(q5)*cos(q6)*cos(q7) - sin(q5)*sin(q7), - cos(q7)*sin(q5) - cos(q5)*cos(q6)*sin(q7), cos(q5)*sin(q6)]
[                           cos(q7)*sin(q6),                            -sin(q6)*sin(q7),        -cos(q6)]
[ cos(q5)*sin(q7) + cos(q6)*cos(q7)*sin(q5),   cos(q5)*cos(q7) - cos(q6)*sin(q5)*sin(q7), sin(q5)*sin(q6)]
*)
METHOD PROTECTED wristIK : BOOL
VAR_IN_OUT CONSTANT
	i_cmdRot :Mat3d;
	i_masterArm :FB_MasterArm;
END_VAR

VAR_OUTPUT
	q5:	LREAL;
	q6:	LREAL;
	q7:	LREAL;
END_VAR

VAR
	invRot :Mat3d;
	jnt4Rotation :Mat3d;
	s5, s7, c5, c7:LREAL;
END_VAR
// calculate wrist joint position
// q6=[-pi/2-45deg, -pi/2+45deg]
IF 1 = i_masterArm.armIdx THEN
	q6:= -ACOS(-i_cmdRot[2,3]);
// q6=[pi/2-45deg, pi/2+45deg]
ELSE
	q6:= ACOS(-i_cmdRot[2,3]);
END_IF

IF q6>GVL_ArmJointParameters.g_maxJntPos[i_masterArm.armIdx, 6] OR q6< GVL_ArmJointParameters.g_minJntPos[i_masterArm.armIdx, 6] THEN
	wristIK:=FALSE;
	RETURN;
END_IF

// q5 = [pi-135deg, pi+135deg]
c5 := i_cmdRot[1,3]/SIN(q6);
s5 := i_cmdRot[3,3]/SIN(q6);
q5:=atan2(s5,c5);
IF q5<GVL_ArmJointParameters.g_minJntPos[1,5] THEN
	q5:=q5+2*PI;
END_IF
IF q5>GVL_ArmJointParameters.g_maxJntPos[1,5]THEN
	wristIK:=FALSE;
	RETURN;
END_IF
c7 := i_cmdRot[2,1]/SIN(q6);
s7 := -i_cmdRot[2,2]/SIN(q6);
q7:=atan2(s7,c7);
wristIK:=true;
END_METHOD

END_FUNCTION_BLOCK

// ---- FBs_StateControllers/FB_StateCtrlReady.TcPOU
// Brief: Master Arm Ready for Master Slave Control
FUNCTION_BLOCK PUBLIC FB_StateCtrlReady EXTENDS FB_MasterArmCtrlBase
VAR_INPUT
END_VAR
VAR_OUTPUT
END_VAR
VAR
	
cmdPos, curPos :Vec7d;
END_VAR

METHOD PUBLIC init : BOOL
VAR_IN_OUT CONSTANT
	i_masterArm	:FB_MasterArm;
END_VAR
VAR_IN_OUT 
	r_masterArmCtrlCmd :ST_ArmCtrlCmds;
END_VAR

VAR
	j:INT;
	maxJntErr:LREAL;
	jntCtrlErr:Vec7d;
END_VAR
// check if to hold the command joint position unchanged
m_holdLastCmds := checkToHoldLastCmds(i_masterArm);

// init
SUPER^.Init(i_masterArm,r_masterArmCtrlCmd);

m_jntOPMode[4] := DriverOPMode_PosTrq;
m_jntOPMode[5] := DriverOPMode_PosTrq;
m_jntOPMode[6] := DriverOPMode_PosTrq;
m_jntOPMode[7] := DriverOPMode_PosTrq;
END_METHOD

END_FUNCTION_BLOCK

// ---- FBs_StateControllers/FB_StateCtrlMasterSlave.TcPOU
// Brief: Master Arm MasterSlave controller
FUNCTION_BLOCK PUBLIC FB_StateCtrlMasterSlave EXTENDS FB_MasterArmCtrlBase
VAR_INPUT
END_VAR
VAR_OUTPUT
END_VAR
VAR
	// joint4 controller
	m_redunJntCtrl : FB_RedunJntControl;
	
	// flag if project joint4 torque to nullspace
	m_nullspaceCtrl : BOOL :=FALSE;
	
	// boundary limit force feedback
	m_boundaryForce : FB_boundaryForceFeedback;
	
	// joint torque for master-slave error
	m_boundaryTrq :Vec7d;
	
	// friction compensation scale
	m_frictionCompScale :LREAL :=0.8;

END_VAR

// override this function in each exact controller
METHOD PROTECTED calcCmdJntPos : BOOL

VAR_IN_OUT CONSTANT
	i_slaveIdx :INT;
	i_shoulderPose :ST_Frame;
	i_masterArm :FB_MasterArm;
	i_slaveStatus :ST_SlaveStatus;
END_VAR
VAR 

END_VAR
IF i_slaveStatus.m_instruStauts[i_slaveIdx].m_type = InstruType_UltrasoundKnifeS OR 
	i_slaveStatus.m_instruStauts[i_slaveIdx].m_type = InstruType_UltrasoundKnifeU THEN
	calcCmdJntPos_USKnife(i_slaveIdx,i_shoulderPose,i_masterArm,i_slaveStatus);
ELSE
	calcCmdJntPos_BasicInstru(i_slaveIdx,i_shoulderPose,i_masterArm,i_slaveStatus);
END_IF
END_METHOD

// override this function in each exact controller
METHOD PROTECTED calcCmdJntPos_BasicInstru : BOOL

VAR_IN_OUT CONSTANT
	i_slaveIdx :INT;
	i_shoulderPose :ST_Frame;
	i_masterArm :FB_MasterArm;
	i_slaveStatus :ST_SlaveStatus;
END_VAR
VAR 

END_VAR
m_cmdJntPos:=i_masterArm.curJntPos;
m_cmdJntVel:=i_masterArm.curJntVel;
m_cmdCartPose:=i_masterArm.curCartPose;
END_METHOD

// override this function in each exact controller
METHOD PROTECTED calcCmdJntPos_USKnife : BOOL

VAR_IN_OUT CONSTANT
	i_slaveIdx :INT;
	i_shoulderPose :ST_Frame;
	i_masterArm :FB_MasterArm;
	i_slaveStatus :ST_SlaveStatus;
END_VAR
VAR CONSTANT
	// orientation tracking parameters
	m_rotTrackKp : LREAL := 200;
	m_maxTrackVel :LREAL := PI;
	m_trackAngThres :LREAL := 2* g_deg2rad;
END_VAR
VAR 
	cartTrackVel :Vec3d;
	i,j : INT;
	invRot :Mat3d;
	cmdRotInView:Mat3d;
	rotT,rotErr :Mat3d;
	angle:LREAL;
	axis:Vec3d;
	
	oriJaco:Mat34;
	oriJt:Mat43;
	oriJJt:Mat3d;
	oriJJtInv:Mat3d;
	oriJPinv:Mat43;
	jntTrackVel:Vec4d;
	JpinvJ, nullJ:Mat4d;
	eye4d :Mat4d := g_eye4d;
	redunCtrlVel :Vec4d;
	jnt4TrackVel :LREAL;
	cmdZAxis, curZAxis :Vec3d;
END_VAR
m_jntOPMode[1] := DriverOPMode_Trq;
m_jntOPMode[2] := DriverOPMode_Trq;
m_jntOPMode[3] := DriverOPMode_Trq;
m_jntOPMode[4] := DriverOPMode_PosTrq;
m_jntOPMode[5] := DriverOPMode_PosTrq;
m_jntOPMode[6] := DriverOPMode_PosTrq;
m_jntOPMode[7] := DriverOPMode_Trq;

// use matched slave arm orientation as target, 
//	and transform from view coordinate to arm coordinate 
cmdRotInView := i_slaveStatus.m_curArmPose[i_slaveIdx].m_rot;
matTranspose(i_shoulderPose.m_rot, invRot);
matMultiply(invRot, cmdRotInView, m_cmdCartPose.m_rot);
m_cmdCartPose.m_pos:= i_masterArm.curCartPose.m_pos;

// first three joints and joint7 is passive control
FOR i:=1 TO 3 DO 
	m_cmdJntPos[i]:=i_masterArm.curJntPos[i];
	m_cmdJntVel[i]:=i_masterArm.curJntVel[i];
END_FOR
m_cmdJntPos[7]:=i_masterArm.curJntPos[7];
m_cmdJntVel[7]:=i_masterArm.curJntVel[7];

// compute cartesian tracking velocity
FOR i:=1 TO 3 DO
	cmdZAxis[i] :=  m_cmdCartPose.m_rot[i,3];
	curZAxis[i] := i_masterArm.simCartPose.m_rot[i,3];
END_FOR
angle := ACOS(LIMIT(-1,vecDot(cmdZAxis,curZAxis),1));
axis := cross(curZAxis, cmdZAxis);
IF ABS(angle)> g_smallAng AND ABS(angle-pi)> g_smallAng THEN
	normalize(axis);
END_IF
vecMultiNum(axis, LIMIT(-m_maxTrackVel, angle*m_rotTrackKp, m_maxTrackVel), cartTrackVel);

// compute pinv of orientation jacobian
FOR i:=1 TO 3 DO
	FOR j:=1 TO 4 DO
		oriJaco[i,j]:=i_masterArm.simJaco[i+3,j+3];
	END_FOR
END_FOR
matTranspose(oriJaco, oriJt);
matMultiply(oriJaco ,oriJt , oriJJt);
invMat3(oriJJt, oriJJtInv);
matMultiply(oriJt, oriJJtInv, oriJPinv);
matMultiVec(oriJpinv, cartTrackVel, jntTrackVel);

// calculate nullspace
matMultiply(oriJPinv, oriJaco, JpinvJ);
matSub(eye4d , JpinvJ, nullJ);

// redundant velocity
jnt4TrackVel:=calcRedunVel(i_masterArm);
redunCtrlVel[1]:=nullJ[1,1]*jnt4TrackVel;
redunCtrlVel[2]:=nullJ[2,1]*jnt4TrackVel;
redunCtrlVel[3]:=nullJ[3,1]*jnt4TrackVel;
redunCtrlVel[4]:=nullJ[4,1]*jnt4TrackVel;

// update final command joint position and velocity
FOR i :=1 TO 3 DO 
	m_cmdJntVel[i+3]:=jntTrackVel[i]+redunCtrlVel[i];
	m_cmdJntPos[i+3]:=m_cmdJntPos[i+3]+m_cmdJntVel[i+3]*g_armCtrlCycleTime;
END_FOR
END_METHOD

// override this function in each exact controller
METHOD PROTECTED calcCmdJntTrq : BOOL

VAR_IN_OUT CONSTANT
	i_slaveIdx :INT;
	i_shoulderPose :ST_Frame;
	i_masterArm :FB_MasterArm;
	i_slaveStatus :ST_SlaveStatus;
END_VAR

VAR 
	nullspaceMat :Mat7d;
	ctrlTrq : Vec7d;
	boundaryTrq :Vec7d;
	withinBoundary :BOOL;
	i :INT;
END_VAR
IF i_slaveStatus.m_instruStauts[i_slaveIdx].m_type = InstruType_UltrasoundKnifeS OR 
	i_slaveStatus.m_instruStauts[i_slaveIdx].m_type = InstruType_UltrasoundKnifeU THEN
	calcCmdJntTrq_USKnife(i_slaveIdx,i_shoulderPose,i_masterArm,i_slaveStatus);
ELSE
	calcCmdJntTrq_BasicInstru(i_slaveIdx,i_shoulderPose,i_masterArm,i_slaveStatus);
END_IF
END_METHOD

// override this function in each exact controller
METHOD PROTECTED calcCmdJntTrq_BasicInstru : BOOL

VAR_IN_OUT CONSTANT
	i_slaveIdx :INT;
	i_shoulderPose :ST_Frame;
	i_masterArm :FB_MasterArm;
	i_slaveStatus :ST_SlaveStatus;
END_VAR

VAR 
	nullspaceMat :Mat7d;
	ctrlTrq : Vec7d;
	boundaryTrq :Vec7d;
	withinBoundary :BOOL;
	i :INT;
END_VAR
// boundary force feedback
m_boundaryTrq :=m_boundaryForce.run(i_slaveIdx, i_shoulderPose, i_masterArm, i_slaveStatus);
withinBoundary := (norm(m_boundaryTrq)<g_smallNum);

// redundant joint4 controller
ctrlTrq := g_zeroVec7d;
ctrlTrq[4] := m_redunJntCtrl.run(i_masterArm, i_followEnable:=withinBoundary);

// project to nullspace
IF m_nullspaceCtrl THEN
	nullspaceMat:=i_masterArm.dynaNullspace;
	matMultiVec(nullspaceMat,ctrlTrq, m_cmdJntTrq);
	vecSelfMultiNum(m_cmdJntTrq, ctrlTrq[4] / m_cmdJntTrq[4]);
ELSE
	m_cmdJntTrq := ctrlTrq;
END_IF

// add friction compensation
FOR i:=1 TO g_mJntNum DO 
	m_cmdJntTrq[i] := m_cmdJntTrq[i] +m_frictionCompScale * i_masterArm.jntFriction[i] + m_boundaryTrq[i];
END_FOR
END_METHOD

// override this function in each exact controller
METHOD PROTECTED calcCmdJntTrq_USKnife : BOOL

VAR_IN_OUT CONSTANT
	i_slaveIdx :INT;
	i_shoulderPose :ST_Frame;
	i_masterArm :FB_MasterArm;
	i_slaveStatus :ST_SlaveStatus;
END_VAR

VAR 
	i :INT;
END_VAR
m_cmdJntTrq :=g_zeroVec7d;
// boundary force feedback
m_boundaryTrq :=m_boundaryForce.run(i_slaveIdx, i_shoulderPose, i_masterArm, i_slaveStatus);
m_cmdJntTrq[7] := m_boundaryTrq[7];
END_METHOD

METHOD PROTECTED calcRedunVel : LREAL
VAR_IN_OUT CONSTANT
	i_masterArm :FB_MasterArm;
END_VAR

VAR 
	// redundant control parameters
	m_jnt4AdjustKp : LREAL :=10;
	m_jnt4MaxVel :LREAL :=pi/3 ;
	m_linearVelLb :LREAL := 0.02;
	m_linearVelUb :LREAL :=0.1;	
	
	j6Bias,j5Bias :LREAL;
	velScale :LREAL;
	linearVel :Vec3d;
	curJntPos : Vec7d;
	jnt4LinkPos :LREAL;
END_VAR
// compute desired joint4 link position
curJntPos :=  i_masterArm.cmdJntPos;
jnt4LinkPos:=i_masterArm.jnt4MotorToLink(curJntPos[2],curJntPos[3],curJntPos[4]);
IF 1= i_masterArm.armIdx THEN
	j6Bias :=curJntPos[6]+PI/2;
ELSE 
	j6Bias := curJntPos[6]-PI/2;
END_IF

// scale based on joint5 position
j5Bias :=  LIMIT (0, ABS(curJntPos[5] -pi), pi/2);
j6Bias := j6Bias * ABS(COS(j5Bias));

// scale based on linear velocity
linearVel[1]:=i_masterArm.curCartTwist[1];
linearVel[2]:=i_masterArm.curCartTwist[2];
linearVel[3]:=i_masterArm.curCartTwist[3];
velScale :=LIMIT(0, (norm(linearVel)-m_linearVelLb)/(m_linearVelUb-m_linearVelLb),1.0);


calcRedunVel := LIMIT(-m_jnt4MaxVel, -j6Bias * m_jnt4AdjustKp * velScale ,m_jnt4MaxVel);

// joint limit
IF (calcRedunVel > 0 AND jnt4LinkPos+calcRedunVel * g_armCtrlCycleTime > GVL_ArmJointParameters.g_maxJntPos[i_masterArm.armIdx,4])
	 OR ( calcRedunVel <0 AND  jnt4LinkPos +calcRedunVel * g_armCtrlCycleTime< GVL_ArmJointParameters.g_minJntPos[i_masterArm.armIdx,4]) THEN
	 calcRedunVel :=0;
END_IF
END_METHOD

METHOD PUBLIC init : BOOL
VAR_IN_OUT CONSTANT
	i_masterArm	:FB_MasterArm;
END_VAR
VAR_IN_OUT 
	r_masterArmCtrlCmd :ST_ArmCtrlCmds;
END_VAR

VAR
	i:INT;
END_VAR
SUPER^.Init(i_masterArm,r_masterArmCtrlCmd);

m_jntOPMode := g_allTrqMode;
//m_jntOPMode := g_allPosMode;

// init controller
m_redunJntCtrl.init(i_masterArm);

// update commands to arm
copyCmds(r_masterArmCtrlCmd);
END_METHOD

END_FUNCTION_BLOCK

// ---- FBs_BasicControllers/FB_RedunJntControl.TcPOU
// Author: Feijian Ni
// Date: 2023.11.22
FUNCTION_BLOCK FB_RedunJntControl
VAR_INPUT
END_VAR
VAR_OUTPUT
END_VAR
VAR
	// joint 6 deviation from center
	m_jnt6Bias :LREAL;
	
	// max target position step 
	m_maxTargetPosStep :LREAL :=10*g_deg2rad;
	
	// static velocity threshold
	m_staticVelThres :LREAL := 60 *g_deg2Rad;
	
	// static threshold of joint bias
	m_staticBiasThres :LREAL := 30 *g_deg2Rad;
	
	// rudundancy track flag
	m_trackFlag :BOOL;
	
	// joint4 track tolerance
	m_joint4TrackTol :LREAL :=1*g_deg2rad;
	
	// orientation nullspace jacobian
	m_oriNullJaco: Mat4d;
	
	// current manipulation velocity
	m_curManipWVel :LREAL :=0;
	
	// joint4 limit buffer
	m_jntLimitBuffer : LREAL :=2.5*g_deg2Rad;
	
	// control paramters for redundant joint4 position control
//	m_redunJntKp: LREAL:=8.0;
//	m_redunJntKd:LREAL:=0.2;
//	m_redunJntKp: LREAL:=3.0;
//	m_redunJntKd:LREAL:=0.1;
	m_redunJntKp: LREAL:=2.5;
	m_redunJntKd:LREAL:=0.05;
	m_redunJntKi:LREAL:=0;
	m_redunJntKiLimit: LREAL:=200;
	m_redunJntCtrlLimit:LREAL:=1000;

	// max vel and acc for joint4 motion
	m_jnt4MaxFollowVel :LREAL :=2*pi;
	m_jnt4MaxFollowAcc :LREAL :=4*pi;
	m_jnt4MinFollowAcc :LREAL :=1.5*pi;
	m_jnt4MinAccVel:LREAL:= 60 *g_deg2Rad;
	m_jnt4MaxAccVel:LREAL:= 150 *g_deg2Rad;
	
	// max acc scale when approaching joint limit
	m_accScaleNearLimit :LREAL;
	m_maxAccScaleNearLimit :LREAL := 1.0;
	m_accScaleBiasLB :LREAL := 30 *g_deg2Rad;
	m_accScaleBiasUB :LREAL := 45 *g_deg2Rad;

